LIN {X 0,Y 488.682,Z 691.608,A -85,B 0,C 180,E1 -6498.445,E2 -6498.445} C_VEL
LIN {X 0,Y 488.641,Z 691.61,A -85,B 0,C 180,E1 -6501.074,E2 -6501.074} C_VEL
LIN {X 0,Y 488.644,Z 691.62,A -85,B 0,C 180,E1 -6503.748,E2 -6503.748} C_VEL
LIN {X 0,Y 488.702,Z 691.604,A -85,B 0,C 180,E1 -6506.475,E2 -6506.475} C_VEL
LIN {X 0,Y 488.669,Z 691.61,A -85,B 0,C 180,E1 -6509.274,E2 -6509.274} C_VEL
LIN {X 0,Y 488.646,Z 691.618,A -85,B 0,C 180,E1 -6512.151,E2 -6512.151} C_VEL
LIN {X 0,Y 488.663,Z 691.609,A -85,B 0,C 180,E1 -6515.12,E2 -6515.12} C_VEL
LIN {X 0,Y 488.636,Z 691.613,A -85,B 0,C 180,E1 -6518.204,E2 -6518.204} C_VEL
LIN {X 0,Y 488.696,Z 691.613,A -85,B 0,C 180,E1 -6520.355,E2 -6520.355} C_VEL
LIN {X 0,Y 488.667,Z 691.611,A -85,B 0,C 180,E1 -6523.657,E2 -6523.657} C_VEL
LIN {X 0,Y 488.67,Z 691.617,A -85,B 0,C 180,E1 -6526.355,E2 -6526.355} C_VEL
LIN {X 0,Y 488.691,Z 691.609,A -85,B 0,C 180,E1 -6529.683,E2 -6529.683} C_VEL
LIN {X 0,Y 488.64,Z 691.619,A -85,B 0,C 180,E1 -6532.284,E2 -6532.284} C_VEL
LIN {X 0,Y 488.691,Z 691.608,A -85,B 0,C 180,E1 -6535.058,E2 -6535.058} C_VEL
LIN {X 0,Y 488.671,Z 691.615,A -85,B 0,C 180,E1 -6538.052,E2 -6538.052} C_VEL
LIN {X 0,Y 488.749,Z 691.808,A -85,B 0,C 180,E1 -6540.178,E2 -6540.178} C_VEL
LIN {X 0,Y 492.403,Z 708.291,A -85,B 0,C 180,E1 -6542.534,E2 -6542.534} C_VEL
LIN {X 0,Y 491.834,Z 726.438,A -85,B 0,C 180,E1 -6544.85,E2 -6544.85} C_VEL
LIN {X 0,Y 491.007,Z 751.019,A -85,B 0,C 180,E1 -6547.938,E2 -6547.938} C_VEL
LIN {X 0,Y 490.21,Z 776.598,A -85,B 0,C 180,E1 -6551.125,E2 -6551.125} C_VEL
LIN {X 0,Y 489.614,Z 797.522,A -85,B 0,C 180,E1 -6553.716,E2 -6553.716} C_VEL
LIN {X 0,Y 491.626,Z 815.137,A -85,B 0,C 180,E1 -6554.041,E2 -6554.041} C_VEL
LIN {X 0,Y 491.033,Z 908.334,A -85,B 0,C 180,E1 -6555.422,E2 -6555.422} C_VEL
LIN {X 0,Y 490.681,Z 921.584,A -85,B 0,C 180,E1 -6555.782,E2 -6555.782} C_VEL
LIN {X 0,Y 490.274,Z 934.931,A -85,B 0,C 180,E1 -6556.325,E2 -6556.325} C_VEL
LIN {X 0,Y 489.962,Z 946.2,A -85,B 0,C 180,E1 -6556.95,E2 -6556.95} C_VEL
LIN {X 0,Y 489.582,Z 957.937,A -85,B 0,C 180,E1 -6557.782,E2 -6557.782} C_VEL
LIN {X 0,Y 489.117,Z 968.518,A -85,B 0,C 180,E1 -6558.716,E2 -6558.716} C_VEL
LIN {X 0,Y 488.829,Z 977.207,A -85,B 0,C 180,E1 -6559.653,E2 -6559.653} C_VEL
LIN {X 0,Y 488.559,Z 985.239,A -85,B 0,C 180,E1 -6560.693,E2 -6560.693} C_VEL
LIN {X 0,Y 488.333,Z 993.106,A -85,B 0,C 180,E1 -6561.94,E2 -6561.94} C_VEL
LIN {X 0,Y 488.136,Z 1000.365,A -85,B 0,C 180,E1 -6563.392,E2 -6563.392} C_VEL
LIN {X 0,Y 488.09,Z 1005.213,A -85,B 0,C 180,E1 -6564.636,E2 -6564.636} C_VEL
LIN {X 0,Y 488.029,Z 1008.92,A -85,B 0,C 180,E1 -6565.877,E2 -6565.877} C_VEL
LIN {X 0,Y 488.027,Z 1010.835,A -85,B 0,C 180,E1 -6566.703,E2 -6566.703} C_VEL
LIN {X 0,Y 487.976,Z 1012.263,A -85,B 0,C 180,E1 -6567.529,E2 -6567.529} C_VEL
LIN {X 0,Y 487.951,Z 1013.283,A -85,B 0,C 180,E1 -6568.355,E2 -6568.355} C_VEL
LIN {X 0,Y 487.913,Z 1013.9,A -85,B 0,C 180,E1 -6569.18,E2 -6569.18} C_VEL
LIN {X 0,Y 487.905,Z 1014.118,A -85,B 0,C 180,E1 -6570.005,E2 -6570.005} C_VEL
LIN {X 0,Y 487.913,Z 1013.893,A -85,B 0,C 180,E1 -6570.831,E2 -6570.831} C_VEL
LIN {X 0,Y 487.952,Z 1013.27,A -85,B 0,C 180,E1 -6571.656,E2 -6571.656} C_VEL
LIN {X 0,Y 487.978,Z 1012.245,A -85,B 0,C 180,E1 -6572.482,E2 -6572.482} C_VEL
LIN {X 0,Y 488.03,Z 1010.81,A -85,B 0,C 180,E1 -6573.307,E2 -6573.307} C_VEL
LIN {X 0,Y 488.022,Z 1007.785,A -85,B 0,C 180,E1 -6574.548,E2 -6574.548} C_VEL
LIN {X 0,Y 488.16,Z 1002.71,A -85,B 0,C 180,E1 -6576.045,E2 -6576.045} C_VEL
LIN {X 0,Y 488.241,Z 996.389,A -85,B 0,C 180,E1 -6577.449,E2 -6577.449} C_VEL
LIN {X 0,Y 488.462,Z 989.326,A -85,B 0,C 180,E1 -6578.694,E2 -6578.694} C_VEL
LIN {X 0,Y 488.713,Z 980.494,A -85,B 0,C 180,E1 -6579.942,E2 -6579.942} C_VEL
LIN {X 0,Y 489.054,Z 971.474,A -85,B 0,C 180,E1 -6580.982,E2 -6580.982} C_VEL
LIN {X 0,Y 489.494,Z 960.399,A -85,B 0,C 180,E1 -6582.021,E2 -6582.021} C_VEL
LIN {X 0,Y 489.843,Z 949.728,A -85,B 0,C 180,E1 -6582.821,E2 -6582.821} C_VEL
LIN {X 0,Y 490.162,Z 937.757,A -85,B 0,C 180,E1 -6583.531,E2 -6583.531} C_VEL
LIN {X 0,Y 490.558,Z 924.976,A -85,B 0,C 180,E1 -6584.101,E2 -6584.101} C_VEL
LIN {X 0,Y 490.92,Z 912.426,A -85,B 0,C 180,E1 -6584.487,E2 -6584.487} C_VEL
LIN {X 0,Y 491.114,Z 896.461,A -85,B 0,C 180,E1 -6584.772,E2 -6584.772} C_VEL
LIN {X 0,Y 491.597,Z 814.634,A -85,B 0,C 180,E1 -6585.967,E2 -6585.967} C_VEL
LIN {X 0,Y 489.604,Z 797.347,A -85,B 0,C 180,E1 -6586.302,E2 -6586.302} C_VEL
LIN {X 0,Y 490.277,Z 773.565,A -85,B 0,C 180,E1 -6589.255,E2 -6589.255} C_VEL
LIN {X 0,Y 491.138,Z 747.424,A -85,B 0,C 180,E1 -6592.51,E2 -6592.51} C_VEL
LIN {X 0,Y 491.835,Z 726.347,A -85,B 0,C 180,E1 -6595.162,E2 -6595.162} C_VEL
LIN {X 0,Y 492.39,Z 707.801,A -85,B 0,C 180,E1 -6597.53,E2 -6597.53} C_VEL
LIN {X 0,Y 488.675,Z 691.615,A -85,B 0,C 180,E1 -6599.87,E2 -6599.87} C_VEL
LIN {X 0,Y 488.684,Z 691.608,A -85,B 0,C 180,E1 -6602.152,E2 -6602.152} C_VEL
LIN {X 0,Y 488.637,Z 691.615,A -85,B 0,C 180,E1 -6605.126,E2 -6605.126} C_VEL
LIN {X 0,Y 488.654,Z 691.613,A -85,B 0,C 180,E1 -6608.206,E2 -6608.206} C_VEL
LIN {X 0,Y 488.657,Z 691.617,A -85,B 0,C 180,E1 -6611.425,E2 -6611.425} C_VEL
LIN {X 0,Y 488.711,Z 691.608,A -85,B 0,C 180,E1 -6614.805,E2 -6614.805} C_VEL
LIN {X 0,Y 488.663,Z 691.616,A -85,B 0,C 180,E1 -6617.471,E2 -6617.471} C_VEL
LIN {X 0,Y 488.719,Z 691.607,A -85,B 0,C 180,E1 -6619.675,E2 -6619.675} C_VEL
LIN {X 0,Y 488.673,Z 691.613,A -85,B 0,C 180,E1 -6622.84,E2 -6622.84} C_VEL
LIN {X 0,Y 488.734,Z 691.603,A -85,B 0,C 180,E1 -6625.887,E2 -6625.887} C_VEL
LIN {X 0,Y 488.704,Z 691.608,A -85,B 0,C 180,E1 -6628.821,E2 -6628.821} C_VEL
LIN {X 0,Y 488.712,Z 691.61,A -85,B 0,C 180,E1 -6631.669,E2 -6631.669} C_VEL
LIN {X 0,Y 488.713,Z 691.606,A -85,B 0,C 180,E1 -6634.442,E2 -6634.442} C_VEL
LIN {X 0,Y 488.734,Z 691.609,A -85,B 0,C 180,E1 -6637.154,E2 -6637.154} C_VEL
LIN {X 0,Y 488.737,Z 691.608,A -85,B 0,C 180,E1 -6639.811,E2 -6639.811} C_VEL
LIN {X 0,Y 488.724,Z 691.606,A -85,B 0,C 180,E1 -6642.423,E2 -6642.423} C_VEL
LIN {X 0,Y 488.782,Z 691.601,A -85,B 0,C 180,E1 -6644.316,E2 -6644.316} C_VEL
LIN {X 0,Y 491.379,Z 699.537,A -85,B 0,C 180,E1 -6644.546,E2 -6644.546} C_VEL
LIN {X 0,Y 490.914,Z 771.943,A -85,B 0,C 180,E1 -6645.729,E2 -6645.729} C_VEL
LIN {X 0,Y 490.85,Z 783.407,A -85,B 0,C 180,E1 -6646.044,E2 -6646.044} C_VEL
LIN {X 0,Y 490.738,Z 793.546,A -85,B 0,C 180,E1 -6646.437,E2 -6646.437} C_VEL
LIN {X 0,Y 490.525,Z 803.477,A -85,B 0,C 180,E1 -6646.936,E2 -6646.936} C_VEL
LIN {X 0,Y 490.338,Z 812.486,A -85,B 0,C 180,E1 -6647.5,E2 -6647.5} C_VEL
LIN {X 0,Y 490.066,Z 821.742,A -85,B 0,C 180,E1 -6648.208,E2 -6648.208} C_VEL
LIN {X 0,Y 489.791,Z 830.671,A -85,B 0,C 180,E1 -6649.04,E2 -6649.04} C_VEL
LIN {X 0,Y 489.536,Z 838.156,A -85,B 0,C 180,E1 -6649.871,E2 -6649.871} C_VEL
LIN {X 0,Y 489.241,Z 845.904,A -85,B 0,C 180,E1 -6650.908,E2 -6650.908} C_VEL
LIN {X 0,Y 489.033,Z 852.313,A -85,B 0,C 180,E1 -6651.945,E2 -6651.945} C_VEL
LIN {X 0,Y 488.829,Z 858.14,A -85,B 0,C 180,E1 -6653.095,E2 -6653.095} C_VEL
LIN {X 0,Y 488.697,Z 862.749,A -85,B 0,C 180,E1 -6654.222,E2 -6654.222} C_VEL
LIN {X 0,Y 488.536,Z 865.607,A -85,B 0,C 180,E1 -6655.048,E2 -6655.048} C_VEL
LIN {X 0,Y 488.424,Z 869.61,A -85,B 0,C 180,E1 -6656.7,E2 -6656.7} C_VEL
LIN {X 0,Y 488.434,Z 871.082,A -85,B 0,C 180,E1 -6657.526,E2 -6657.526} C_VEL
LIN {X 0,Y 488.379,Z 872.611,A -85,B 0,C 180,E1 -6659.175,E2 -6659.175} C_VEL
LIN {X 0,Y 488.346,Z 872.803,A -85,B 0,C 180,E1 -6660,E2 -6660} C_VEL
LIN {X 0,Y 488.322,Z 872.573,A -85,B 0,C 180,E1 -6660.825,E2 -6660.825} C_VEL
LIN {X 0,Y 488.287,Z 870.905,A -85,B 0,C 180,E1 -6662.475,E2 -6662.475} C_VEL
LIN {X 0,Y 488.448,Z 867.553,A -85,B 0,C 180,E1 -6664.126,E2 -6664.126} C_VEL
LIN {X 0,Y 488.527,Z 863.892,A -85,B 0,C 180,E1 -6665.366,E2 -6665.366} C_VEL
LIN {X 0,Y 488.748,Z 859.084,A -85,B 0,C 180,E1 -6666.606,E2 -6666.606} C_VEL
LIN {X 0,Y 488.857,Z 854.178,A -85,B 0,C 180,E1 -6667.642,E2 -6667.642} C_VEL
LIN {X 0,Y 489.102,Z 848.229,A -85,B 0,C 180,E1 -6668.678,E2 -6668.678} C_VEL
LIN {X 0,Y 489.325,Z 841.043,A -85,B 0,C 180,E1 -6669.716,E2 -6669.716} C_VEL
LIN {X 0,Y 489.586,Z 832.308,A -85,B 0,C 180,E1 -6670.755,E2 -6670.755} C_VEL
LIN {X 0,Y 489.9,Z 823.903,A -85,B 0,C 180,E1 -6671.586,E2 -6671.586} C_VEL
LIN {X 0,Y 490.138,Z 815.105,A -85,B 0,C 180,E1 -6672.315,E2 -6672.315} C_VEL
LIN {X 0,Y 490.391,Z 805.826,A -85,B 0,C 180,E1 -6672.95,E2 -6672.95} C_VEL
LIN {X 0,Y 490.643,Z 795.612,A -85,B 0,C 180,E1 -6673.513,E2 -6673.513} C_VEL
LIN {X 0,Y 490.802,Z 785.306,A -85,B 0,C 180,E1 -6673.957,E2 -6673.957} C_VEL
LIN {X 0,Y 490.895,Z 774.608,A -85,B 0,C 180,E1 -6674.298,E2 -6674.298} C_VEL
LIN {X 0,Y 491.019,Z 762.121,A -85,B 0,C 180,E1 -6674.559,E2 -6674.559} C_VEL
LIN {X 0,Y 491.415,Z 699.602,A -85,B 0,C 180,E1 -6675.532,E2 -6675.532} C_VEL
LIN {X 0,Y 488.767,Z 691.601,A -85,B 0,C 180,E1 -6675.76,E2 -6675.76} C_VEL
LIN {X 0,Y 488.76,Z 691.604,A -85,B 0,C 180,E1 -6678.442,E2 -6678.442} C_VEL
LIN {X 0,Y 488.72,Z 691.607,A -85,B 0,C 180,E1 -6681.07,E2 -6681.07} C_VEL
LIN {X 0,Y 488.685,Z 691.607,A -85,B 0,C 180,E1 -6683.746,E2 -6683.746} C_VEL
LIN {X 0,Y 488.728,Z 691.609,A -85,B 0,C 180,E1 -6686.925,E2 -6686.925} C_VEL
LIN {X 0,Y 488.737,Z 691.602,A -85,B 0,C 180,E1 -6690.219,E2 -6690.219} C_VEL
LIN {X 0,Y 488.725,Z 691.603,A -85,B 0,C 180,E1 -6693.478,E2 -6693.478} C_VEL
LIN {X 0,Y 488.687,Z 691.608,A -85,B 0,C 180,E1 -6696.351,E2 -6696.351} C_VEL
LIN {X 0,Y 488.708,Z 691.608,A -85,B 0,C 180,E1 -6699.254,E2 -6699.254} C_VEL
LIN {X 0,Y 488.683,Z 691.608,A -85,B 0,C 180,E1 -6702.527,E2 -6702.527} C_VEL
LIN {X 0,Y 488.713,Z 691.609,A -85,B 0,C 180,E1 -6705.195,E2 -6705.195} C_VEL
LIN {X 0,Y 488.677,Z 691.609,A -85,B 0,C 180,E1 -6708.577,E2 -6708.577} C_VEL
LIN {X 0,Y 488.7,Z 691.61,A -85,B 0,C 180,E1 -6710.948,E2 -6710.948} C_VEL
LIN {X 0,Y 488.651,Z 691.611,A -85,B 0,C 180,E1 -6713.447,E2 -6713.447} C_VEL
LIN {X 0,Y 488.007,Z 691.694,A -85,B 0,C 180,E1 -6714.134,E2 -6714.134} C_VEL
LIN {X 0,Y 485.168,Z 692.051,A -85,B 0,C 180,E1 -6715.251,E2 -6715.251} C_VEL
LIN {X 0,Y 482.758,Z 692.346,A -85,B 0,C 180,E1 -6716.152,E2 -6716.152} C_VEL
LIN {X 0,Y 481.726,Z 692.477,A -85,B 0,C 180,E1 -6716.847,E2 -6716.847} C_VEL
LIN {X 0,Y 481.644,Z 692.487,A -85,B 0,C 180,E1 -6717.083,E2 -6717.083} C_VEL
LIN {X 0,Y 481.613,Z 692.487,A -85,B 0,C 180,E1 -6720.25,E2 -6720.25} C_VEL
LIN {X 0,Y 481.642,Z 692.49,A -85,B 0,C 180,E1 -6723.102,E2 -6723.102} C_VEL
LIN {X 0,Y 481.633,Z 692.488,A -85,B 0,C 180,E1 -6725.88,E2 -6725.88} C_VEL
LIN {X 0,Y 481.666,Z 692.488,A -85,B 0,C 180,E1 -6729.04,E2 -6729.04} C_VEL
LIN {X 0,Y 481.665,Z 692.486,A -85,B 0,C 180,E1 -6732.152,E2 -6732.152} C_VEL
LIN {X 0,Y 481.658,Z 692.489,A -85,B 0,C 180,E1 -6733.9,E2 -6733.9} C_VEL
LIN {X 0,Y 485.021,Z 702.116,A -85,B 0,C 180,E1 -6734.18,E2 -6734.18} C_VEL
LIN {X 0,Y 484.543,Z 773.549,A -85,B 0,C 180,E1 -6735.264,E2 -6735.264} C_VEL
LIN {X 0,Y 484.601,Z 786.67,A -85,B 0,C 180,E1 -6735.642,E2 -6735.642} C_VEL
LIN {X 0,Y 484.417,Z 798.704,A -85,B 0,C 180,E1 -6736.146,E2 -6736.146} C_VEL
LIN {X 0,Y 484.157,Z 810.293,A -85,B 0,C 180,E1 -6736.798,E2 -6736.798} C_VEL
LIN {X 0,Y 483.754,Z 821.579,A -85,B 0,C 180,E1 -6737.621,E2 -6737.621} C_VEL
LIN {X 0,Y 483.388,Z 831.928,A -85,B 0,C 180,E1 -6738.57,E2 -6738.57} C_VEL
LIN {X 0,Y 483.057,Z 840.367,A -85,B 0,C 180,E1 -6739.517,E2 -6739.517} C_VEL
LIN {X 0,Y 482.687,Z 848.134,A -85,B 0,C 180,E1 -6740.567,E2 -6740.567} C_VEL
LIN {X 0,Y 482.29,Z 855.831,A -85,B 0,C 180,E1 -6741.848,E2 -6741.848} C_VEL
LIN {X 0,Y 482.153,Z 861.483,A -85,B 0,C 180,E1 -6743.022,E2 -6743.022} C_VEL
LIN {X 0,Y 481.851,Z 867.263,A -85,B 0,C 180,E1 -6744.555,E2 -6744.555} C_VEL
LIN {X 0,Y 481.625,Z 870.803,A -85,B 0,C 180,E1 -6745.811,E2 -6745.811} C_VEL
LIN {X 0,Y 481.532,Z 872.63,A -85,B 0,C 180,E1 -6746.648,E2 -6746.648} C_VEL
LIN {X 0,Y 481.529,Z 874.001,A -85,B 0,C 180,E1 -6747.485,E2 -6747.485} C_VEL
LIN {X 0,Y 481.486,Z 875.581,A -85,B 0,C 180,E1 -6749.158,E2 -6749.158} C_VEL
LIN {X 0,Y 481.469,Z 875.817,A -85,B 0,C 180,E1 -6749.994,E2 -6749.994} C_VEL
LIN {X 0,Y 481.565,Z 875.065,A -85,B 0,C 180,E1 -6751.667,E2 -6751.667} C_VEL
LIN {X 0,Y 481.523,Z 872.825,A -85,B 0,C 180,E1 -6753.341,E2 -6753.341} C_VEL
LIN {X 0,Y 481.685,Z 870.022,A -85,B 0,C 180,E1 -6754.597,E2 -6754.597} C_VEL
LIN {X 0,Y 481.908,Z 866.215,A -85,B 0,C 180,E1 -6755.853,E2 -6755.853} C_VEL
LIN {X 0,Y 482.113,Z 860.745,A -85,B 0,C 180,E1 -6757.242,E2 -6757.242} C_VEL
LIN {X 0,Y 482.412,Z 853.941,A -85,B 0,C 180,E1 -6758.582,E2 -6758.582} C_VEL
LIN {X 0,Y 482.814,Z 845.931,A -85,B 0,C 180,E1 -6759.842,E2 -6759.842} C_VEL
LIN {X 0,Y 483.164,Z 837.724,A -85,B 0,C 180,E1 -6760.894,E2 -6760.894} C_VEL
LIN {X 0,Y 483.542,Z 827.573,A -85,B 0,C 180,E1 -6761.947,E2 -6761.947} C_VEL
LIN {X 0,Y 484.001,Z 817.128,A -85,B 0,C 180,E1 -6762.814,E2 -6762.814} C_VEL
LIN {X 0,Y 484.302,Z 805.369,A -85,B 0,C 180,E1 -6763.592,E2 -6763.592} C_VEL
LIN {X 0,Y 484.494,Z 792.885,A -85,B 0,C 180,E1 -6764.211,E2 -6764.211} C_VEL
LIN {X 0,Y 484.657,Z 779.801,A -85,B 0,C 180,E1 -6764.667,E2 -6764.667} C_VEL
LIN {X 0,Y 484.662,Z 767.477,A -85,B 0,C 180,E1 -6764.935,E2 -6764.935} C_VEL
LIN {X 0,Y 485.002,Z 701.859,A -85,B 0,C 180,E1 -6765.916,E2 -6765.916} C_VEL
LIN {X 0,Y 481.693,Z 692.485,A -85,B 0,C 180,E1 -6766.185,E2 -6766.185} C_VEL
LIN {X 0,Y 481.693,Z 692.488,A -85,B 0,C 180,E1 -6768.715,E2 -6768.715} C_VEL
LIN {X 0,Y 481.626,Z 692.489,A -85,B 0,C 180,E1 -6771.388,E2 -6771.388} C_VEL
LIN {X 0,Y 481.628,Z 692.485,A -85,B 0,C 180,E1 -6774.108,E2 -6774.108} C_VEL
LIN {X 0,Y 481.689,Z 692.485,A -85,B 0,C 180,E1 -6777.125,E2 -6777.125} C_VEL
LIN {X 0,Y 481.649,Z 692.485,A -85,B 0,C 180,E1 -6779.734,E2 -6779.734} C_VEL
LIN {X 0,Y 481.639,Z 692.487,A -85,B 0,C 180,E1 -6782.668,E2 -6782.668} C_VEL
LIN {X 0,Y 481.605,Z 692.494,A -85,B 0,C 180,E1 -6785.703,E2 -6785.703} C_VEL
LIN {X 0,Y 481.673,Z 692.48,A -85,B 0,C 180,E1 -6789.347,E2 -6789.347} C_VEL
LIN {X 0,Y 481.631,Z 692.489,A -85,B 0,C 180,E1 -6792.151,E2 -6792.151} C_VEL
LIN {X 0,Y 481.613,Z 692.482,A -85,B 0,C 180,E1 -6794.451,E2 -6794.451} C_VEL
LIN {X 0,Y 481.639,Z 692.482,A -85,B 0,C 180,E1 -6796.84,E2 -6796.84} C_VEL
LIN {X 0,Y 481.661,Z 692.486,A -85,B 0,C 180,E1 -6800.058,E2 -6800.058} C_VEL
LIN {X 0,Y 481.574,Z 692.495,A -85,B 0,C 180,E1 -6803.37,E2 -6803.37} C_VEL
LIN {X 0,Y 481.649,Z 692.487,A -85,B 0,C 180,E1 -6806.325,E2 -6806.325} C_VEL
LIN {X 0,Y 481.6,Z 692.49,A -85,B 0,C 180,E1 -6809.41,E2 -6809.41} C_VEL
LIN {X 0,Y 481.637,Z 692.49,A -85,B 0,C 180,E1 -6812.164,E2 -6812.164} C_VEL
LIN {X 0,Y 481.653,Z 692.482,A -85,B 0,C 180,E1 -6814.966,E2 -6814.966} C_VEL
LIN {X 0,Y 481.585,Z 692.49,A -85,B 0,C 180,E1 -6817.701,E2 -6817.701} C_VEL
LIN {X 0,Y 481.636,Z 692.493,A -85,B 0,C 180,E1 -6820.39,E2 -6820.39} C_VEL
LIN {X 0,Y 481.621,Z 692.486,A -85,B 0,C 180,E1 -6823.031,E2 -6823.031} C_VEL
LIN {X 0,Y 481.631,Z 692.486,A -85,B 0,C 180,E1 -6825.637,E2 -6825.637} C_VEL
LIN {X 0,Y 481.723,Z 692.477,A -85,B 0,C 180,E1 -6828.214,E2 -6828.214} C_VEL
LIN {X 0,Y 481.695,Z 692.479,A -85,B 0,C 180,E1 -6831.61,E2 -6831.61} C_VEL
LIN {X 0,Y 481.756,Z 692.472,A -85,B 0,C 180,E1 -6834.139,E2 -6834.139} C_VEL
LIN {X 0,Y 481.859,Z 692.46,A -85,B 0,C 180,E1 -6837.492,E2 -6837.492} C_VEL
LIN {X 0,Y 481.859,Z 692.459,A -85,B 0,C 180,E1 -6840,E2 -6840} C_VEL
LIN {X 0,Y 481.859,Z 692.457,A -85,B 0,C 180,E1 -6842.508,E2 -6842.508} C_VEL
LIN {X 0,Y 481.756,Z 692.473,A -85,B 0,C 180,E1 -6845.861,E2 -6845.861} C_VEL
LIN {X 0,Y 481.695,Z 692.476,A -85,B 0,C 180,E1 -6848.389,E2 -6848.389} C_VEL
LIN {X 0,Y 481.722,Z 692.478,A -85,B 0,C 180,E1 -6851.786,E2 -6851.786} C_VEL
LIN {X 0,Y 481.675,Z 692.486,A -85,B 0,C 180,E1 -6855.226,E2 -6855.226} C_VEL
LIN {X 0,Y 481.64,Z 692.485,A -85,B 0,C 180,E1 -6858.725,E2 -6858.725} C_VEL
LIN {X 0,Y 481.583,Z 692.493,A -85,B 0,C 180,E1 -6861.398,E2 -6861.398} C_VEL
LIN {X 0,Y 481.627,Z 692.488,A -85,B 0,C 180,E1 -6864.116,E2 -6864.116} C_VEL
LIN {X 0,Y 481.686,Z 692.478,A -85,B 0,C 180,E1 -6867.145,E2 -6867.145} C_VEL
LIN {X 0,Y 481.626,Z 692.493,A -85,B 0,C 180,E1 -6869.745,E2 -6869.745} C_VEL
LIN {X 0,Y 481.613,Z 692.489,A -85,B 0,C 180,E1 -6872.679,E2 -6872.679} C_VEL
LIN {X 0,Y 481.584,Z 692.495,A -85,B 0,C 180,E1 -6875.714,E2 -6875.714} C_VEL
LIN {X 0,Y 481.673,Z 692.475,A -85,B 0,C 180,E1 -6879.361,E2 -6879.361} C_VEL
LIN {X 0,Y 481.624,Z 692.495,A -85,B 0,C 180,E1 -6882.163,E2 -6882.163} C_VEL
LIN {X 0,Y 481.611,Z 692.495,A -85,B 0,C 180,E1 -6884.463,E2 -6884.463} C_VEL
LIN {X 0,Y 481.643,Z 692.484,A -85,B 0,C 180,E1 -6886.852,E2 -6886.852} C_VEL
LIN {X 0,Y 481.647,Z 692.489,A -85,B 0,C 180,E1 -6890.067,E2 -6890.067} C_VEL
LIN {X 0,Y 481.589,Z 692.493,A -85,B 0,C 180,E1 -6893.26,E2 -6893.26} C_VEL
LIN {X 0,Y 481.675,Z 692.478,A -85,B 0,C 180,E1 -6896.337,E2 -6896.337} C_VEL
LIN {X 0,Y 481.714,Z 692.67,A -85,B 0,C 180,E1 -6899.939,E2 -6899.939} C_VEL
LIN {X 0,Y 485.499,Z 709.671,A -85,B 0,C 180,E1 -6902.413,E2 -6902.413} C_VEL
LIN {X 0,Y 484.924,Z 727.286,A -85,B 0,C 180,E1 -6904.696,E2 -6904.696} C_VEL
LIN {X 0,Y 484.001,Z 753.142,A -85,B 0,C 180,E1 -6907.992,E2 -6907.992} C_VEL
LIN {X 0,Y 483.107,Z 779.604,A -85,B 0,C 180,E1 -6911.342,E2 -6911.342} C_VEL
LIN {X 0,Y 482.611,Z 796.441,A -85,B 0,C 180,E1 -6913.466,E2 -6913.466} C_VEL
LIN {X 0,Y 484.76,Z 816.114,A -85,B 0,C 180,E1 -6913.839,E2 -6913.839} C_VEL
LIN {X 0,Y 484.146,Z 907.318,A -85,B 0,C 180,E1 -6915.21,E2 -6915.21} C_VEL
LIN {X 0,Y 483.776,Z 920.567,A -85,B 0,C 180,E1 -6915.574,E2 -6915.574} C_VEL
LIN {X 0,Y 483.344,Z 933.913,A -85,B 0,C 180,E1 -6916.125,E2 -6916.125} C_VEL
LIN {X 0,Y 482.958,Z 945.493,A -85,B 0,C 180,E1 -6916.778,E2 -6916.778} C_VEL
LIN {X 0,Y 482.547,Z 957.589,A -85,B 0,C 180,E1 -6917.656,E2 -6917.656} C_VEL
LIN {X 0,Y 482.037,Z 968.556,A -85,B 0,C 180,E1 -6918.655,E2 -6918.655} C_VEL
LIN {X 0,Y 481.721,Z 977.898,A -85,B 0,C 180,E1 -6919.711,E2 -6919.711} C_VEL
LIN {X 0,Y 481.42,Z 987.018,A -85,B 0,C 180,E1 -6920.977,E2 -6920.977} C_VEL
LIN {X 0,Y 481.206,Z 994.377,A -85,B 0,C 180,E1 -6922.242,E2 -6922.242} C_VEL
LIN {X 0,Y 481.07,Z 1001.048,A -85,B 0,C 180,E1 -6923.704,E2 -6923.704} C_VEL
LIN {X 0,Y 480.997,Z 1005.548,A -85,B 0,C 180,E1 -6924.976,E2 -6924.976} C_VEL
LIN {X 0,Y 480.974,Z 1007.911,A -85,B 0,C 180,E1 -6925.816,E2 -6925.816} C_VEL
LIN {X 0,Y 480.982,Z 1009.828,A -85,B 0,C 180,E1 -6926.655,E2 -6926.655} C_VEL
LIN {X 0,Y 480.938,Z 1011.258,A -85,B 0,C 180,E1 -6927.493,E2 -6927.493} C_VEL
LIN {X 0,Y 480.916,Z 1012.279,A -85,B 0,C 180,E1 -6928.331,E2 -6928.331} C_VEL
LIN {X 0,Y 480.883,Z 1012.897,A -85,B 0,C 180,E1 -6929.168,E2 -6929.168} C_VEL
LIN {X 0,Y 480.876,Z 1013.115,A -85,B 0,C 180,E1 -6930.006,E2 -6930.006} C_VEL
LIN {X 0,Y 480.883,Z 1012.89,A -85,B 0,C 180,E1 -6930.843,E2 -6930.843} C_VEL
LIN {X 0,Y 480.917,Z 1012.266,A -85,B 0,C 180,E1 -6931.68,E2 -6931.68} C_VEL
LIN {X 0,Y 480.939,Z 1011.24,A -85,B 0,C 180,E1 -6932.518,E2 -6932.518} C_VEL
LIN {X 0,Y 480.985,Z 1009.803,A -85,B 0,C 180,E1 -6933.356,E2 -6933.356} C_VEL
LIN {X 0,Y 480.977,Z 1006.776,A -85,B 0,C 180,E1 -6934.615,E2 -6934.615} C_VEL
LIN {X 0,Y 481.092,Z 1002.699,A -85,B 0,C 180,E1 -6935.874,E2 -6935.874} C_VEL
LIN {X 0,Y 481.158,Z 996.41,A -85,B 0,C 180,E1 -6937.348,E2 -6937.348} C_VEL
LIN {X 0,Y 481.35,Z 989.569,A -85,B 0,C 180,E1 -6938.612,E2 -6938.612} C_VEL
LIN {X 0,Y 481.597,Z 981.098,A -85,B 0,C 180,E1 -6939.878,E2 -6939.878} C_VEL
LIN {X 0,Y 481.943,Z 972.436,A -85,B 0,C 180,E1 -6940.933,E2 -6940.933} C_VEL
LIN {X 0,Y 482.392,Z 961.768,A -85,B 0,C 180,E1 -6941.987,E2 -6941.987} C_VEL
LIN {X 0,Y 482.828,Z 949.931,A -85,B 0,C 180,E1 -6942.926,E2 -6942.926} C_VEL
LIN {X 0,Y 483.19,Z 937.742,A -85,B 0,C 180,E1 -6943.676,E2 -6943.676} C_VEL
LIN {X 0,Y 483.606,Z 925.269,A -85,B 0,C 180,E1 -6944.254,E2 -6944.254} C_VEL
LIN {X 0,Y 483.995,Z 912.471,A -85,B 0,C 180,E1 -6944.672,E2 -6944.672} C_VEL
LIN {X 0,Y 484.203,Z 899.035,A -85,B 0,C 180,E1 -6944.934,E2 -6944.934} C_VEL
LIN {X 0,Y 484.757,Z 815.001,A -85,B 0,C 180,E1 -6946.178,E2 -6946.178} C_VEL
LIN {X 0,Y 482.58,Z 796.32,A -85,B 0,C 180,E1 -6946.546,E2 -6946.546} C_VEL
LIN {X 0,Y 483.285,Z 773.894,A -85,B 0,C 180,E1 -6949.383,E2 -6949.383} C_VEL
LIN {X 0,Y 484.171,Z 748.254,A -85,B 0,C 180,E1 -6952.627,E2 -6952.627} C_VEL
LIN {X 0,Y 484.929,Z 727.191,A -85,B 0,C 180,E1 -6955.316,E2 -6955.316} C_VEL
LIN {X 0,Y 485.52,Z 709.573,A -85,B 0,C 180,E1 -6957.598,E2 -6957.598} C_VEL
LIN {X 0,Y 481.634,Z 692.492,A -85,B 0,C 180,E1 -6960.11,E2 -6960.11} C_VEL
LIN {X 0,Y 481.626,Z 692.487,A -85,B 0,C 180,E1 -6962.682,E2 -6962.682} C_VEL
LIN {X 0,Y 481.58,Z 692.489,A -85,B 0,C 180,E1 -6965.718,E2 -6965.718} C_VEL
LIN {X 0,Y 481.629,Z 692.492,A -85,B 0,C 180,E1 -6968.867,E2 -6968.867} C_VEL
LIN {X 0,Y 481.624,Z 692.488,A -85,B 0,C 180,E1 -6971.909,E2 -6971.909} C_VEL
LIN {X 0,Y 481.647,Z 692.485,A -85,B 0,C 180,E1 -6974.463,E2 -6974.463} C_VEL
LIN {X 0,Y 481.627,Z 692.49,A -85,B 0,C 180,E1 -6976.858,E2 -6976.858} C_VEL
LIN {X 0,Y 481.671,Z 692.482,A -85,B 0,C 180,E1 -6980.059,E2 -6980.059} C_VEL
LIN {X 0,Y 481.631,Z 692.494,A -85,B 0,C 180,E1 -6983.38,E2 -6983.38} C_VEL
LIN {X 0,Y 481.686,Z 692.48,A -85,B 0,C 180,E1 -6986.328,E2 -6986.328} C_VEL
LIN {X 0,Y 481.662,Z 692.489,A -85,B 0,C 180,E1 -6989.419,E2 -6989.419} C_VEL
LIN {X 0,Y 481.67,Z 692.484,A -85,B 0,C 180,E1 -6992.166,E2 -6992.166} C_VEL
LIN {X 0,Y 481.691,Z 692.484,A -85,B 0,C 180,E1 -6994.968,E2 -6994.968} C_VEL
LIN {X 0,Y 481.661,Z 692.489,A -85,B 0,C 180,E1 -6997.705,E2 -6997.705} C_VEL
LIN {X 0,Y 481.717,Z 692.479,A -85,B 0,C 180,E1 -7000.393,E2 -7000.393} C_VEL
LIN {X 0,Y 481.688,Z 692.486,A -85,B 0,C 180,E1 -7003.034,E2 -7003.034} C_VEL
LIN {X 0,Y 481.727,Z 692.481,A -85,B 0,C 180,E1 -7004.067,E2 -7004.067} C_VEL
LIN {X 0,Y 484.579,Z 700.942,A -85,B 0,C 180,E1 -7004.328,E2 -7004.328} C_VEL
LIN {X 0,Y 484.029,Z 773.443,A -85,B 0,C 180,E1 -7005.549,E2 -7005.549} C_VEL
LIN {X 0,Y 483.946,Z 784.76,A -85,B 0,C 180,E1 -7005.868,E2 -7005.868} C_VEL
LIN {X 0,Y 483.884,Z 795.369,A -85,B 0,C 180,E1 -7006.295,E2 -7006.295} C_VEL
LIN {X 0,Y 483.63,Z 805.455,A -85,B 0,C 180,E1 -7006.819,E2 -7006.819} C_VEL
LIN {X 0,Y 483.414,Z 814.468,A -85,B 0,C 180,E1 -7007.404,E2 -7007.404} C_VEL
LIN {X 0,Y 483.126,Z 823.784,A -85,B 0,C 180,E1 -7008.143,E2 -7008.143} C_VEL
LIN {X 0,Y 482.885,Z 831.592,A -85,B 0,C 180,E1 -7008.881,E2 -7008.881} C_VEL
LIN {X 0,Y 482.615,Z 839.118,A -85,B 0,C 180,E1 -7009.724,E2 -7009.724} C_VEL
LIN {X 0,Y 482.302,Z 846.898,A -85,B 0,C 180,E1 -7010.776,E2 -7010.776} C_VEL
LIN {X 0,Y 482.078,Z 853.333,A -85,B 0,C 180,E1 -7011.828,E2 -7011.828} C_VEL
LIN {X 0,Y 481.877,Z 859.169,A -85,B 0,C 180,E1 -7012.993,E2 -7012.993} C_VEL
LIN {X 0,Y 481.731,Z 863.8,A -85,B 0,C 180,E1 -7014.139,E2 -7014.139} C_VEL
LIN {X 0,Y 481.542,Z 866.665,A -85,B 0,C 180,E1 -7014.976,E2 -7014.976} C_VEL
LIN {X 0,Y 481.416,Z 870.674,A -85,B 0,C 180,E1 -7016.652,E2 -7016.652} C_VEL
LIN {X 0,Y 481.427,Z 872.141,A -85,B 0,C 180,E1 -7017.49,E2 -7017.49} C_VEL
LIN {X 0,Y 481.372,Z 873.659,A -85,B 0,C 180,E1 -7019.163,E2 -7019.163} C_VEL
LIN {X 0,Y 481.339,Z 873.839,A -85,B 0,C 180,E1 -7020,E2 -7020} C_VEL
LIN {X 0,Y 481.32,Z 873.595,A -85,B 0,C 180,E1 -7020.837,E2 -7020.837} C_VEL
LIN {X 0,Y 481.265,Z 871.904,A -85,B 0,C 180,E1 -7022.511,E2 -7022.511} C_VEL
LIN {X 0,Y 481.432,Z 868.506,A -85,B 0,C 180,E1 -7024.186,E2 -7024.186} C_VEL
LIN {X 0,Y 481.528,Z 864.809,A -85,B 0,C 180,E1 -7025.444,E2 -7025.444} C_VEL
LIN {X 0,Y 481.765,Z 859.966,A -85,B 0,C 180,E1 -7026.702,E2 -7026.702} C_VEL
LIN {X 0,Y 481.891,Z 855.009,A -85,B 0,C 180,E1 -7027.753,E2 -7027.753} C_VEL
LIN {X 0,Y 482.125,Z 849.013,A -85,B 0,C 180,E1 -7028.804,E2 -7028.804} C_VEL
LIN {X 0,Y 482.385,Z 841.769,A -85,B 0,C 180,E1 -7029.857,E2 -7029.857} C_VEL
LIN {X 0,Y 482.607,Z 834.946,A -85,B 0,C 180,E1 -7030.7,E2 -7030.7} C_VEL
LIN {X 0,Y 482.934,Z 825.668,A -85,B 0,C 180,E1 -7031.649,E2 -7031.649} C_VEL
LIN {X 0,Y 483.209,Z 817.022,A -85,B 0,C 180,E1 -7032.388,E2 -7032.388} C_VEL
LIN {X 0,Y 483.467,Z 806.876,A -85,B 0,C 180,E1 -7033.098,E2 -7033.098} C_VEL
LIN {X 0,Y 483.718,Z 796.935,A -85,B 0,C 180,E1 -7033.656,E2 -7033.656} C_VEL
LIN {X 0,Y 483.909,Z 786.02,A -85,B 0,C 180,E1 -7034.133,E2 -7034.133} C_VEL
LIN {X 0,Y 484.012,Z 775.252,A -85,B 0,C 180,E1 -7034.479,E2 -7034.479} C_VEL
LIN {X 0,Y 484.133,Z 762.67,A -85,B 0,C 180,E1 -7034.744,E2 -7034.744} C_VEL
LIN {X 0,Y 484.557,Z 701.038,A -85,B 0,C 180,E1 -7035.725,E2 -7035.725} C_VEL
LIN {X 0,Y 481.716,Z 692.48,A -85,B 0,C 180,E1 -7035.979,E2 -7035.979} C_VEL
LIN {X 0,Y 481.721,Z 692.483,A -85,B 0,C 180,E1 -7038.721,E2 -7038.721} C_VEL
LIN {X 0,Y 481.658,Z 692.484,A -85,B 0,C 180,E1 -7041.394,E2 -7041.394} C_VEL
LIN {X 0,Y 481.665,Z 692.483,A -85,B 0,C 180,E1 -7044.114,E2 -7044.114} C_VEL
LIN {X 0,Y 481.7,Z 692.481,A -85,B 0,C 180,E1 -7047.124,E2 -7047.124} C_VEL
LIN {X 0,Y 481.687,Z 692.479,A -85,B 0,C 180,E1 -7049.741,E2 -7049.741} C_VEL
LIN {X 0,Y 481.667,Z 692.487,A -85,B 0,C 180,E1 -7052.675,E2 -7052.675} C_VEL
LIN {X 0,Y 481.645,Z 692.484,A -85,B 0,C 180,E1 -7055.709,E2 -7055.709} C_VEL
LIN {X 0,Y 481.681,Z 692.487,A -85,B 0,C 180,E1 -7058.858,E2 -7058.858} C_VEL
LIN {X 0,Y 481.641,Z 692.483,A -85,B 0,C 180,E1 -7062.162,E2 -7062.162} C_VEL
LIN {X 0,Y 481.67,Z 692.48,A -85,B 0,C 180,E1 -7064.457,E2 -7064.457} C_VEL
LIN {X 0,Y 481.63,Z 692.485,A -85,B 0,C 180,E1 -7067.834,E2 -7067.834} C_VEL
LIN {X 0,Y 481.661,Z 692.483,A -85,B 0,C 180,E1 -7070.654,E2 -7070.654} C_VEL
LIN {X 0,Y 481.617,Z 692.49,A -85,B 0,C 180,E1 -7073.442,E2 -7073.442} C_VEL
LIN {X 0,Y 481.687,Z 692.477,A -85,B 0,C 180,E1 -7076.324,E2 -7076.324} C_VEL
LIN {X 0,Y 481.644,Z 692.487,A -85,B 0,C 180,E1 -7077.083,E2 -7077.083} C_VEL
LIN {X 0,Y 480.979,Z 692.574,A -85,B 0,C 180,E1 -7077.781,E2 -7077.781} C_VEL
LIN {X 0,Y 478.111,Z 692.928,A -85,B 0,C 180,E1 -7078.914,E2 -7078.914} C_VEL
LIN {X 0,Y 475.69,Z 693.226,A -85,B 0,C 180,E1 -7079.827,E2 -7079.827} C_VEL
LIN {X 0,Y 474.662,Z 693.354,A -85,B 0,C 180,E1 -7080.533,E2 -7080.533} C_VEL
LIN {X 0,Y 474.584,Z 693.365,A -85,B 0,C 180,E1 -7080.772,E2 -7080.772} C_VEL
LIN {X 0,Y 474.569,Z 693.37,A -85,B 0,C 180,E1 -7083.619,E2 -7083.619} C_VEL
LIN {X 0,Y 474.611,Z 693.363,A -85,B 0,C 180,E1 -7086.649,E2 -7086.649} C_VEL
LIN {X 0,Y 474.629,Z 693.366,A -85,B 0,C 180,E1 -7089.179,E2 -7089.179} C_VEL
LIN {X 0,Y 474.626,Z 693.364,A -85,B 0,C 180,E1 -7091.879,E2 -7091.879} C_VEL
LIN {X 0,Y 474.615,Z 693.368,A -85,B 0,C 180,E1 -7093.655,E2 -7093.655} C_VEL
LIN {X 0,Y 478.274,Z 704.058,A -85,B 0,C 180,E1 -7093.965,E2 -7093.965} C_VEL
LIN {X 0,Y 477.746,Z 774.571,A -85,B 0,C 180,E1 -7095.05,E2 -7095.05} C_VEL
LIN {X 0,Y 477.794,Z 787.686,A -85,B 0,C 180,E1 -7095.433,E2 -7095.433} C_VEL
LIN {X 0,Y 477.595,Z 799.716,A -85,B 0,C 180,E1 -7095.944,E2 -7095.944} C_VEL
LIN {X 0,Y 477.318,Z 811.297,A -85,B 0,C 180,E1 -7096.605,E2 -7096.605} C_VEL
LIN {X 0,Y 476.893,Z 822.587,A -85,B 0,C 180,E1 -7097.44,E2 -7097.44} C_VEL
LIN {X 0,Y 476.503,Z 832.935,A -85,B 0,C 180,E1 -7098.402,E2 -7098.402} C_VEL
LIN {X 0,Y 476.152,Z 841.373,A -85,B 0,C 180,E1 -7099.363,E2 -7099.363} C_VEL
LIN {X 0,Y 475.759,Z 849.139,A -85,B 0,C 180,E1 -7100.429,E2 -7100.429} C_VEL
LIN {X 0,Y 475.335,Z 856.836,A -85,B 0,C 180,E1 -7101.728,E2 -7101.728} C_VEL
LIN {X 0,Y 475.18,Z 862.486,A -85,B 0,C 180,E1 -7102.919,E2 -7102.919} C_VEL
LIN {X 0,Y 474.865,Z 868.266,A -85,B 0,C 180,E1 -7104.474,E2 -7104.474} C_VEL
LIN {X 0,Y 474.616,Z 871.807,A -85,B 0,C 180,E1 -7105.749,E2 -7105.749} C_VEL
LIN {X 0,Y 474.515,Z 873.633,A -85,B 0,C 180,E1 -7106.598,E2 -7106.598} C_VEL
LIN {X 0,Y 474.514,Z 875.003,A -85,B 0,C 180,E1 -7107.448,E2 -7107.448} C_VEL
LIN {X 0,Y 474.467,Z 876.583,A -85,B 0,C 180,E1 -7109.146,E2 -7109.146} C_VEL
LIN {X 0,Y 474.449,Z 876.818,A -85,B 0,C 180,E1 -7109.994,E2 -7109.994} C_VEL
LIN {X 0,Y 474.551,Z 876.065,A -85,B 0,C 180,E1 -7111.692,E2 -7111.692} C_VEL
LIN {X 0,Y 474.506,Z 873.827,A -85,B 0,C 180,E1 -7113.391,E2 -7113.391} C_VEL
LIN {X 0,Y 474.679,Z 871.023,A -85,B 0,C 180,E1 -7114.665,E2 -7114.665} C_VEL
LIN {X 0,Y 474.925,Z 867.216,A -85,B 0,C 180,E1 -7115.94,E2 -7115.94} C_VEL
LIN {X 0,Y 475.142,Z 861.744,A -85,B 0,C 180,E1 -7117.349,E2 -7117.349} C_VEL
LIN {X 0,Y 475.466,Z 854.941,A -85,B 0,C 180,E1 -7118.708,E2 -7118.708} C_VEL
LIN {X 0,Y 475.894,Z 846.93,A -85,B 0,C 180,E1 -7119.986,E2 -7119.986} C_VEL
LIN {X 0,Y 476.291,Z 838.719,A -85,B 0,C 180,E1 -7121.053,E2 -7121.053} C_VEL
LIN {X 0,Y 476.669,Z 828.571,A -85,B 0,C 180,E1 -7122.122,E2 -7122.122} C_VEL
LIN {X 0,Y 477.15,Z 818.124,A -85,B 0,C 180,E1 -7123.002,E2 -7123.002} C_VEL
LIN {X 0,Y 477.473,Z 806.364,A -85,B 0,C 180,E1 -7123.791,E2 -7123.791} C_VEL
LIN {X 0,Y 477.675,Z 793.879,A -85,B 0,C 180,E1 -7124.418,E2 -7124.418} C_VEL
LIN {X 0,Y 477.844,Z 780.791,A -85,B 0,C 180,E1 -7124.881,E2 -7124.881} C_VEL
LIN {X 0,Y 477.841,Z 768.456,A -85,B 0,C 180,E1 -7125.154,E2 -7125.154} C_VEL
LIN {X 0,Y 478.238,Z 703.504,A -85,B 0,C 180,E1 -7126.137,E2 -7126.137} C_VEL
LIN {X 0,Y 474.629,Z 693.368,A -85,B 0,C 180,E1 -7126.433,E2 -7126.433} C_VEL
LIN {X 0,Y 474.647,Z 693.366,A -85,B 0,C 180,E1 -7129.004,E2 -7129.004} C_VEL
LIN {X 0,Y 474.569,Z 693.366,A -85,B 0,C 180,E1 -7131.722,E2 -7131.722} C_VEL
LIN {X 0,Y 474.606,Z 693.362,A -85,B 0,C 180,E1 -7134.488,E2 -7134.488} C_VEL
LIN {X 0,Y 474.647,Z 693.36,A -85,B 0,C 180,E1 -7137.326,E2 -7137.326} C_VEL
LIN {X 0,Y 474.575,Z 693.364,A -85,B 0,C 180,E1 -7140.223,E2 -7140.223} C_VEL
LIN {X 0,Y 474.61,Z 693.368,A -85,B 0,C 180,E1 -7143.213,E2 -7143.213} C_VEL
LIN {X 0,Y 474.554,Z 693.368,A -85,B 0,C 180,E1 -7146.317,E2 -7146.317} C_VEL
LIN {X 0,Y 474.61,Z 693.366,A -85,B 0,C 180,E1 -7149.644,E2 -7149.644} C_VEL
LIN {X 0,Y 474.607,Z 693.363,A -85,B 0,C 180,E1 -7152.924,E2 -7152.924} C_VEL
LIN {X 0,Y 474.569,Z 693.366,A -85,B 0,C 180,E1 -7155.89,E2 -7155.89} C_VEL
LIN {X 0,Y 474.595,Z 693.364,A -85,B 0,C 180,E1 -7159.032,E2 -7159.032} C_VEL
LIN {X 0,Y 474.566,Z 693.37,A -85,B 0,C 180,E1 -7161.697,E2 -7161.697} C_VEL
LIN {X 0,Y 474.571,Z 693.365,A -85,B 0,C 180,E1 -7164.721,E2 -7164.721} C_VEL
LIN {X 0,Y 474.578,Z 693.368,A -85,B 0,C 180,E1 -7167.783,E2 -7167.783} C_VEL
LIN {X 0,Y 474.567,Z 693.362,A -85,B 0,C 180,E1 -7170.878,E2 -7170.878} C_VEL
LIN {X 0,Y 474.6,Z 693.363,A -85,B 0,C 180,E1 -7173.625,E2 -7173.625} C_VEL
LIN {X 0,Y 474.567,Z 693.367,A -85,B 0,C 180,E1 -7176.637,E2 -7176.637} C_VEL
LIN {X 0,Y 474.585,Z 693.368,A -85,B 0,C 180,E1 -7180.086,E2 -7180.086} C_VEL
LIN {X 0,Y 474.58,Z 693.366,A -85,B 0,C 180,E1 -7182.772,E2 -7182.772} C_VEL
LIN {X 0,Y 474.587,Z 693.364,A -85,B 0,C 180,E1 -7185.419,E2 -7185.419} C_VEL
LIN {X 0,Y 474.665,Z 693.354,A -85,B 0,C 180,E1 -7188.036,E2 -7188.036} C_VEL
LIN {X 0,Y 474.66,Z 693.356,A -85,B 0,C 180,E1 -7191.485,E2 -7191.485} C_VEL
LIN {X 0,Y 474.716,Z 693.349,A -85,B 0,C 180,E1 -7194.052,E2 -7194.052} C_VEL
LIN {X 0,Y 474.826,Z 693.336,A -85,B 0,C 180,E1 -7197.455,E2 -7197.455} C_VEL
LIN {X 0,Y 474.831,Z 693.335,A -85,B 0,C 180,E1 -7200,E2 -7200} C_VEL
LIN {X 0,Y 474.826,Z 693.333,A -85,B 0,C 180,E1 -7202.545,E2 -7202.545} C_VEL
LIN {X 0,Y 474.716,Z 693.35,A -85,B 0,C 180,E1 -7205.948,E2 -7205.948} C_VEL
LIN {X 0,Y 474.66,Z 693.353,A -85,B 0,C 180,E1 -7208.515,E2 -7208.515} C_VEL
LIN {X 0,Y 474.665,Z 693.356,A -85,B 0,C 180,E1 -7211.963,E2 -7211.963} C_VEL
LIN {X 0,Y 474.63,Z 693.362,A -85,B 0,C 180,E1 -7215.78,E2 -7215.78} C_VEL
LIN {X 0,Y 474.593,Z 693.365,A -85,B 0,C 180,E1 -7219.013,E2 -7219.013} C_VEL
LIN {X 0,Y 474.527,Z 693.375,A -85,B 0,C 180,E1 -7221.732,E2 -7221.732} C_VEL
LIN {X 0,Y 474.607,Z 693.36,A -85,B 0,C 180,E1 -7224.496,E2 -7224.496} C_VEL
LIN {X 0,Y 474.633,Z 693.358,A -85,B 0,C 180,E1 -7227.343,E2 -7227.343} C_VEL
LIN {X 0,Y 474.55,Z 693.366,A -85,B 0,C 180,E1 -7230.817,E2 -7230.817} C_VEL
LIN {X 0,Y 474.578,Z 693.37,A -85,B 0,C 180,E1 -7233.989,E2 -7233.989} C_VEL
LIN {X 0,Y 474.519,Z 693.371,A -85,B 0,C 180,E1 -7236.905,E2 -7236.905} C_VEL
LIN {X 0,Y 474.616,Z 693.355,A -85,B 0,C 180,E1 -7239.659,E2 -7239.659} C_VEL
LIN {X 0,Y 474.602,Z 693.363,A -85,B 0,C 180,E1 -7242.936,E2 -7242.936} C_VEL
LIN {X 0,Y 474.571,Z 693.369,A -85,B 0,C 180,E1 -7245.902,E2 -7245.902} C_VEL
LIN {X 0,Y 474.604,Z 693.365,A -85,B 0,C 180,E1 -7249.044,E2 -7249.044} C_VEL
LIN {X 0,Y 474.576,Z 693.366,A -85,B 0,C 180,E1 -7251.71,E2 -7251.71} C_VEL
LIN {X 0,Y 474.592,Z 693.369,A -85,B 0,C 180,E1 -7254.733,E2 -7254.733} C_VEL
LIN {X 0,Y 474.603,Z 693.367,A -85,B 0,C 180,E1 -7257.794,E2 -7257.794} C_VEL
LIN {X 0,Y 474.633,Z 693.483,A -85,B 0,C 180,E1 -7259.684,E2 -7259.684} C_VEL
LIN {X 0,Y 478.525,Z 710.522,A -85,B 0,C 180,E1 -7262.214,E2 -7262.214} C_VEL
LIN {X 0,Y 478.365,Z 720.389,A -85,B 0,C 180,E1 -7263.527,E2 -7263.527} C_VEL
LIN {X 0,Y 477.215,Z 749.179,A -85,B 0,C 180,E1 -7267.265,E2 -7267.265} C_VEL
LIN {X 0,Y 476.226,Z 775.842,A -85,B 0,C 180,E1 -7270.694,E2 -7270.694} C_VEL
LIN {X 0,Y 475.613,Z 795.82,A -85,B 0,C 180,E1 -7273.229,E2 -7273.229} C_VEL
LIN {X 0,Y 477.913,Z 817.076,A -85,B 0,C 180,E1 -7273.631,E2 -7273.631} C_VEL
LIN {X 0,Y 477.256,Z 906.301,A -85,B 0,C 180,E1 -7274.991,E2 -7274.991} C_VEL
LIN {X 0,Y 476.886,Z 919.551,A -85,B 0,C 180,E1 -7275.361,E2 -7275.361} C_VEL
LIN {X 0,Y 476.435,Z 932.897,A -85,B 0,C 180,E1 -7275.92,E2 -7275.92} C_VEL
LIN {X 0,Y 476.002,Z 944.15,A -85,B 0,C 180,E1 -7276.56,E2 -7276.56} C_VEL
LIN {X 0,Y 475.533,Z 955.91,A -85,B 0,C 180,E1 -7277.418,E2 -7277.418} C_VEL
LIN {X 0,Y 475.082,Z 966.475,A -85,B 0,C 180,E1 -7278.378,E2 -7278.378} C_VEL
LIN {X 0,Y 474.754,Z 975.165,A -85,B 0,C 180,E1 -7279.343,E2 -7279.343} C_VEL
LIN {X 0,Y 474.465,Z 983.2,A -85,B 0,C 180,E1 -7280.414,E2 -7280.414} C_VEL
LIN {X 0,Y 474.19,Z 991.067,A -85,B 0,C 180,E1 -7281.698,E2 -7281.698} C_VEL
LIN {X 0,Y 474.058,Z 996.469,A -85,B 0,C 180,E1 -7282.767,E2 -7282.767} C_VEL
LIN {X 0,Y 474.024,Z 1001.723,A -85,B 0,C 180,E1 -7284.049,E2 -7284.049} C_VEL
LIN {X 0,Y 473.93,Z 1005.799,A -85,B 0,C 180,E1 -7285.328,E2 -7285.328} C_VEL
LIN {X 0,Y 473.938,Z 1008.821,A -85,B 0,C 180,E1 -7286.605,E2 -7286.605} C_VEL
LIN {X 0,Y 473.898,Z 1010.253,A -85,B 0,C 180,E1 -7287.456,E2 -7287.456} C_VEL
LIN {X 0,Y 473.881,Z 1011.274,A -85,B 0,C 180,E1 -7288.306,E2 -7288.306} C_VEL
LIN {X 0,Y 473.853,Z 1011.894,A -85,B 0,C 180,E1 -7289.156,E2 -7289.156} C_VEL
LIN {X 0,Y 473.848,Z 1012.113,A -85,B 0,C 180,E1 -7290.006,E2 -7290.006} C_VEL
LIN {X 0,Y 473.853,Z 1011.887,A -85,B 0,C 180,E1 -7290.855,E2 -7290.855} C_VEL
LIN {X 0,Y 473.882,Z 1011.262,A -85,B 0,C 180,E1 -7291.705,E2 -7291.705} C_VEL
LIN {X 0,Y 473.9,Z 1010.235,A -85,B 0,C 180,E1 -7292.555,E2 -7292.555} C_VEL
LIN {X 0,Y 473.941,Z 1008.796,A -85,B 0,C 180,E1 -7293.406,E2 -7293.406} C_VEL
LIN {X 0,Y 473.934,Z 1005.769,A -85,B 0,C 180,E1 -7294.684,E2 -7294.684} C_VEL
LIN {X 0,Y 474.033,Z 1001.687,A -85,B 0,C 180,E1 -7295.962,E2 -7295.962} C_VEL
LIN {X 0,Y 474.104,Z 995.395,A -85,B 0,C 180,E1 -7297.458,E2 -7297.458} C_VEL
LIN {X 0,Y 474.3,Z 988.552,A -85,B 0,C 180,E1 -7298.741,E2 -7298.741} C_VEL
LIN {X 0,Y 474.541,Z 980.076,A -85,B 0,C 180,E1 -7300.027,E2 -7300.027} C_VEL
LIN {X 0,Y 474.923,Z 971.416,A -85,B 0,C 180,E1 -7301.096,E2 -7301.096} C_VEL
LIN {X 0,Y 475.39,Z 961.005,A -85,B 0,C 180,E1 -7302.143,E2 -7302.143} C_VEL
LIN {X 0,Y 475.801,Z 950.207,A -85,B 0,C 180,E1 -7303.023,E2 -7303.023} C_VEL
LIN {X 0,Y 476.162,Z 938.677,A -85,B 0,C 180,E1 -7303.773,E2 -7303.773} C_VEL
LIN {X 0,Y 476.632,Z 926.875,A -85,B 0,C 180,E1 -7304.358,E2 -7304.358} C_VEL
LIN {X 0,Y 477.07,Z 914.226,A -85,B 0,C 180,E1 -7304.808,E2 -7304.808} C_VEL
LIN {X 0,Y 477.315,Z 901.379,A -85,B 0,C 180,E1 -7305.1,E2 -7305.1} C_VEL
LIN {X 0,Y 477.881,Z 815.191,A -85,B 0,C 180,E1 -7306.399,E2 -7306.399} C_VEL
LIN {X 0,Y 475.583,Z 795.462,A -85,B 0,C 180,E1 -7306.781,E2 -7306.781} C_VEL
LIN {X 0,Y 476.357,Z 771.678,A -85,B 0,C 180,E1 -7309.841,E2 -7309.841} C_VEL
LIN {X 0,Y 477.218,Z 749.073,A -85,B 0,C 180,E1 -7312.747,E2 -7312.747} C_VEL
LIN {X 0,Y 478.054,Z 726.269,A -85,B 0,C 180,E1 -7315.706,E2 -7315.706} C_VEL
LIN {X 0,Y 478.589,Z 710.923,A -85,B 0,C 180,E1 -7317.728,E2 -7317.728} C_VEL
LIN {X 0,Y 474.591,Z 693.37,A -85,B 0,C 180,E1 -7320.354,E2 -7320.354} C_VEL
LIN {X 0,Y 474.58,Z 693.369,A -85,B 0,C 180,E1 -7323.229,E2 -7323.229} C_VEL
LIN {X 0,Y 474.555,Z 693.364,A -85,B 0,C 180,E1 -7326.331,E2 -7326.331} C_VEL
LIN {X 0,Y 474.611,Z 693.365,A -85,B 0,C 180,E1 -7329.553,E2 -7329.553} C_VEL
LIN {X 0,Y 474.58,Z 693.369,A -85,B 0,C 180,E1 -7332.942,E2 -7332.942} C_VEL
LIN {X 0,Y 474.595,Z 693.364,A -85,B 0,C 180,E1 -7335.893,E2 -7335.893} C_VEL
LIN {X 0,Y 474.614,Z 693.365,A -85,B 0,C 180,E1 -7339.047,E2 -7339.047} C_VEL
LIN {X 0,Y 474.607,Z 693.365,A -85,B 0,C 180,E1 -7341.709,E2 -7341.709} C_VEL
LIN {X 0,Y 474.631,Z 693.361,A -85,B 0,C 180,E1 -7344.726,E2 -7344.726} C_VEL
LIN {X 0,Y 474.649,Z 693.359,A -85,B 0,C 180,E1 -7347.789,E2 -7347.789} C_VEL
LIN {X 0,Y 474.616,Z 693.365,A -85,B 0,C 180,E1 -7350.891,E2 -7350.891} C_VEL
LIN {X 0,Y 474.617,Z 693.367,A -85,B 0,C 180,E1 -7353.626,E2 -7353.626} C_VEL
LIN {X 0,Y 474.649,Z 693.359,A -85,B 0,C 180,E1 -7356.643,E2 -7356.643} C_VEL
LIN {X 0,Y 474.667,Z 693.359,A -85,B 0,C 180,E1 -7360.09,E2 -7360.09} C_VEL
LIN {X 0,Y 474.649,Z 693.361,A -85,B 0,C 180,E1 -7362.774,E2 -7362.774} C_VEL
LIN {X 0,Y 474.682,Z 693.359,A -85,B 0,C 180,E1 -7363.815,E2 -7363.815} C_VEL
LIN {X 0,Y 477.806,Z 702.397,A -85,B 0,C 180,E1 -7364.105,E2 -7364.105} C_VEL
LIN {X 0,Y 477.183,Z 774.056,A -85,B 0,C 180,E1 -7365.337,E2 -7365.337} C_VEL
LIN {X 0,Y 477.124,Z 785.536,A -85,B 0,C 180,E1 -7365.662,E2 -7365.662} C_VEL
LIN {X 0,Y 477.036,Z 796.243,A -85,B 0,C 180,E1 -7366.094,E2 -7366.094} C_VEL
LIN {X 0,Y 476.778,Z 806.503,A -85,B 0,C 180,E1 -7366.633,E2 -7366.633} C_VEL
LIN {X 0,Y 476.554,Z 815.455,A -85,B 0,C 180,E1 -7367.22,E2 -7367.22} C_VEL
LIN {X 0,Y 476.245,Z 824.804,A -85,B 0,C 180,E1 -7367.969,E2 -7367.969} C_VEL
LIN {X 0,Y 475.995,Z 832.618,A -85,B 0,C 180,E1 -7368.718,E2 -7368.718} C_VEL
LIN {X 0,Y 475.716,Z 840.148,A -85,B 0,C 180,E1 -7369.573,E2 -7369.573} C_VEL
LIN {X 0,Y 475.393,Z 847.927,A -85,B 0,C 180,E1 -7370.641,E2 -7370.641} C_VEL
LIN {X 0,Y 475.154,Z 854.363,A -85,B 0,C 180,E1 -7371.708,E2 -7371.708} C_VEL
LIN {X 0,Y 474.923,Z 860.122,A -85,B 0,C 180,E1 -7372.87,E2 -7372.87} C_VEL
LIN {X 0,Y 474.762,Z 864.851,A -85,B 0,C 180,E1 -7374.052,E2 -7374.052} C_VEL
LIN {X 0,Y 474.548,Z 867.723,A -85,B 0,C 180,E1 -7374.902,E2 -7374.902} C_VEL
LIN {X 0,Y 474.409,Z 871.737,A -85,B 0,C 180,E1 -7376.603,E2 -7376.603} C_VEL
LIN {X 0,Y 474.42,Z 873.201,A -85,B 0,C 180,E1 -7377.453,E2 -7377.453} C_VEL
LIN {X 0,Y 474.363,Z 874.706,A -85,B 0,C 180,E1 -7379.151,E2 -7379.151} C_VEL
LIN {X 0,Y 474.33,Z 874.877,A -85,B 0,C 180,E1 -7380,E2 -7380} C_VEL
LIN {X 0,Y 474.316,Z 874.619,A -85,B 0,C 180,E1 -7380.849,E2 -7380.849} C_VEL
LIN {X 0,Y 474.243,Z 872.902,A -85,B 0,C 180,E1 -7382.548,E2 -7382.548} C_VEL
LIN {X 0,Y 474.416,Z 869.461,A -85,B 0,C 180,E1 -7384.248,E2 -7384.248} C_VEL
LIN {X 0,Y 474.529,Z 865.726,A -85,B 0,C 180,E1 -7385.524,E2 -7385.524} C_VEL
LIN {X 0,Y 474.784,Z 860.84,A -85,B 0,C 180,E1 -7386.801,E2 -7386.801} C_VEL
LIN {X 0,Y 474.92,Z 855.837,A -85,B 0,C 180,E1 -7387.868,E2 -7387.868} C_VEL
LIN {X 0,Y 475.167,Z 849.789,A -85,B 0,C 180,E1 -7388.934,E2 -7388.934} C_VEL
LIN {X 0,Y 475.427,Z 842.488,A -85,B 0,C 180,E1 -7390.003,E2 -7390.003} C_VEL
LIN {X 0,Y 475.683,Z 835.596,A -85,B 0,C 180,E1 -7390.858,E2 -7390.858} C_VEL
LIN {X 0,Y 476.015,Z 826.241,A -85,B 0,C 180,E1 -7391.821,E2 -7391.821} C_VEL
LIN {X 0,Y 476.289,Z 817.502,A -85,B 0,C 180,E1 -7392.571,E2 -7392.571} C_VEL
LIN {X 0,Y 476.554,Z 807.858,A -85,B 0,C 180,E1 -7393.253,E2 -7393.253} C_VEL
LIN {X 0,Y 476.83,Z 797.134,A -85,B 0,C 180,E1 -7393.858,E2 -7393.858} C_VEL
LIN {X 0,Y 477.024,Z 786.727,A -85,B 0,C 180,E1 -7394.314,E2 -7394.314} C_VEL
LIN {X 0,Y 477.127,Z 775.878,A -85,B 0,C 180,E1 -7394.665,E2 -7394.665} C_VEL
LIN {X 0,Y 477.252,Z 763.202,A -85,B 0,C 180,E1 -7394.934,E2 -7394.934} C_VEL
LIN {X 0,Y 477.737,Z 702.496,A -85,B 0,C 180,E1 -7395.923,E2 -7395.923} C_VEL
LIN {X 0,Y 474.676,Z 693.358,A -85,B 0,C 180,E1 -7396.179,E2 -7396.179} C_VEL
LIN {X 0,Y 474.675,Z 693.358,A -85,B 0,C 180,E1 -7399.01,E2 -7399.01} C_VEL
LIN {X 0,Y 474.601,Z 693.361,A -85,B 0,C 180,E1 -7401.728,E2 -7401.728} C_VEL
LIN {X 0,Y 474.643,Z 693.361,A -85,B 0,C 180,E1 -7404.494,E2 -7404.494} C_VEL
LIN {X 0,Y 474.653,Z 693.357,A -85,B 0,C 180,E1 -7407.323,E2 -7407.323} C_VEL
LIN {X 0,Y 474.616,Z 693.361,A -85,B 0,C 180,E1 -7410.23,E2 -7410.23} C_VEL
LIN {X 0,Y 474.63,Z 693.362,A -85,B 0,C 180,E1 -7413.221,E2 -7413.221} C_VEL
LIN {X 0,Y 474.599,Z 693.362,A -85,B 0,C 180,E1 -7416.323,E2 -7416.323} C_VEL
LIN {X 0,Y 474.637,Z 693.358,A -85,B 0,C 180,E1 -7419.547,E2 -7419.547} C_VEL
LIN {X 0,Y 474.601,Z 693.36,A -85,B 0,C 180,E1 -7422.23,E2 -7422.23} C_VEL
LIN {X 0,Y 474.63,Z 693.361,A -85,B 0,C 180,E1 -7425.296,E2 -7425.296} C_VEL
LIN {X 0,Y 474.607,Z 693.359,A -85,B 0,C 180,E1 -7428.209,E2 -7428.209} C_VEL
LIN {X 0,Y 474.632,Z 693.357,A -85,B 0,C 180,E1 -7430.449,E2 -7430.449} C_VEL
LIN {X 0,Y 474.583,Z 693.364,A -85,B 0,C 180,E1 -7433.672,E2 -7433.672} C_VEL
LIN {X 0,Y 474.623,Z 693.36,A -85,B 0,C 180,E1 -7436.774,E2 -7436.774} C_VEL
LIN {X 0,Y 474.564,Z 693.367,A -85,B 0,C 180,E1 -7439.763,E2 -7439.763} C_VEL
LIN {X 0,Y 474.584,Z 693.365,A -85,B 0,C 180,E1 -7440.772,E2 -7440.772} C_VEL
LIN {X 0,Y 473.944,Z 693.45,A -85,B 0,C 180,E1 -7441.481,E2 -7441.481} C_VEL
LIN {X 0,Y 471.128,Z 693.799,A -85,B 0,C 180,E1 -7442.632,E2 -7442.632} C_VEL
LIN {X 0,Y 468.719,Z 694.099,A -85,B 0,C 180,E1 -7443.56,E2 -7443.56} C_VEL
LIN {X 0,Y 467.66,Z 694.227,A -85,B 0,C 180,E1 -7444.277,E2 -7444.277} C_VEL
LIN {X 0,Y 467.561,Z 694.24,A -85,B 0,C 180,E1 -7444.52,E2 -7444.52} C_VEL
LIN {X 0,Y 467.564,Z 694.244,A -85,B 0,C 180,E1 -7446.991,E2 -7446.991} C_VEL
LIN {X 0,Y 467.548,Z 694.246,A -85,B 0,C 180,E1 -7449.769,E2 -7449.769} C_VEL
LIN {X 0,Y 467.58,Z 694.241,A -85,B 0,C 180,E1 -7452.501,E2 -7452.501} C_VEL
LIN {X 0,Y 467.574,Z 694.246,A -85,B 0,C 180,E1 -7453.401,E2 -7453.401} C_VEL
LIN {X 0,Y 471.39,Z 705.058,A -85,B 0,C 180,E1 -7453.724,E2 -7453.724} C_VEL
LIN {X 0,Y 470.965,Z 775.592,A -85,B 0,C 180,E1 -7454.83,E2 -7454.83} C_VEL
LIN {X 0,Y 470.989,Z 788.702,A -85,B 0,C 180,E1 -7455.217,E2 -7455.217} C_VEL
LIN {X 0,Y 470.778,Z 800.728,A -85,B 0,C 180,E1 -7455.736,E2 -7455.736} C_VEL
LIN {X 0,Y 470.485,Z 812.3,A -85,B 0,C 180,E1 -7456.406,E2 -7456.406} C_VEL
LIN {X 0,Y 470.036,Z 823.595,A -85,B 0,C 180,E1 -7457.254,E2 -7457.254} C_VEL
LIN {X 0,Y 469.621,Z 833.942,A -85,B 0,C 180,E1 -7458.23,E2 -7458.23} C_VEL
LIN {X 0,Y 469.25,Z 842.378,A -85,B 0,C 180,E1 -7459.205,E2 -7459.205} C_VEL
LIN {X 0,Y 468.834,Z 850.144,A -85,B 0,C 180,E1 -7460.286,E2 -7460.286} C_VEL
LIN {X 0,Y 468.381,Z 857.841,A -85,B 0,C 180,E1 -7461.604,E2 -7461.604} C_VEL
LIN {X 0,Y 468.208,Z 863.489,A -85,B 0,C 180,E1 -7462.812,E2 -7462.812} C_VEL
LIN {X 0,Y 467.88,Z 869.269,A -85,B 0,C 180,E1 -7464.392,E2 -7464.392} C_VEL
LIN {X 0,Y 467.607,Z 872.811,A -85,B 0,C 180,E1 -7465.685,E2 -7465.685} C_VEL
LIN {X 0,Y 467.499,Z 874.637,A -85,B 0,C 180,E1 -7466.547,E2 -7466.547} C_VEL
LIN {X 0,Y 467.498,Z 876.006,A -85,B 0,C 180,E1 -7467.41,E2 -7467.41} C_VEL
LIN {X 0,Y 467.448,Z 877.585,A -85,B 0,C 180,E1 -7469.133,E2 -7469.133} C_VEL
LIN {X 0,Y 467.428,Z 877.82,A -85,B 0,C 180,E1 -7469.994,E2 -7469.994} C_VEL
LIN {X 0,Y 467.536,Z 877.066,A -85,B 0,C 180,E1 -7471.717,E2 -7471.717} C_VEL
LIN {X 0,Y 467.49,Z 874.829,A -85,B 0,C 180,E1 -7473.442,E2 -7473.442} C_VEL
LIN {X 0,Y 467.675,Z 872.025,A -85,B 0,C 180,E1 -7474.735,E2 -7474.735} C_VEL
LIN {X 0,Y 467.942,Z 868.216,A -85,B 0,C 180,E1 -7476.029,E2 -7476.029} C_VEL
LIN {X 0,Y 468.173,Z 862.744,A -85,B 0,C 180,E1 -7477.459,E2 -7477.459} C_VEL
LIN {X 0,Y 468.521,Z 855.941,A -85,B 0,C 180,E1 -7478.838,E2 -7478.838} C_VEL
LIN {X 0,Y 468.977,Z 847.929,A -85,B 0,C 180,E1 -7480.135,E2 -7480.135} C_VEL
LIN {X 0,Y 469.404,Z 839.717,A -85,B 0,C 180,E1 -7481.217,E2 -7481.217} C_VEL
LIN {X 0,Y 469.8,Z 829.569,A -85,B 0,C 180,E1 -7482.302,E2 -7482.302} C_VEL
LIN {X 0,Y 470.305,Z 819.121,A -85,B 0,C 180,E1 -7483.194,E2 -7483.194} C_VEL
LIN {X 0,Y 470.651,Z 807.359,A -85,B 0,C 180,E1 -7483.994,E2 -7483.994} C_VEL
LIN {X 0,Y 470.865,Z 794.872,A -85,B 0,C 180,E1 -7484.631,E2 -7484.631} C_VEL
LIN {X 0,Y 471.036,Z 781.782,A -85,B 0,C 180,E1 -7485.101,E2 -7485.101} C_VEL
LIN {X 0,Y 471.031,Z 769.436,A -85,B 0,C 180,E1 -7485.378,E2 -7485.378} C_VEL
LIN {X 0,Y 471.456,Z 705.074,A -85,B 0,C 180,E1 -7486.366,E2 -7486.366} C_VEL
LIN {X 0,Y 467.59,Z 694.246,A -85,B 0,C 180,E1 -7486.687,E2 -7486.687} C_VEL
LIN {X 0,Y 467.606,Z 694.24,A -85,B 0,C 180,E1 -7489.301,E2 -7489.301} C_VEL
LIN {X 0,Y 467.514,Z 694.244,A -85,B 0,C 180,E1 -7492.067,E2 -7492.067} C_VEL
LIN {X 0,Y 467.547,Z 694.244,A -85,B 0,C 180,E1 -7494.882,E2 -7494.882} C_VEL
LIN {X 0,Y 467.589,Z 694.235,A -85,B 0,C 180,E1 -7497.762,E2 -7497.762} C_VEL
LIN {X 0,Y 467.537,Z 694.247,A -85,B 0,C 180,E1 -7501.038,E2 -7501.038} C_VEL
LIN {X 0,Y 467.555,Z 694.239,A -85,B 0,C 180,E1 -7504.236,E2 -7504.236} C_VEL
LIN {X 0,Y 467.511,Z 694.251,A -85,B 0,C 180,E1 -7507.18,E2 -7507.18} C_VEL
LIN {X 0,Y 467.555,Z 694.242,A -85,B 0,C 180,E1 -7510.256,E2 -7510.256} C_VEL
LIN {X 0,Y 467.575,Z 694.238,A -85,B 0,C 180,E1 -7512.565,E2 -7512.565} C_VEL
LIN {X 0,Y 467.525,Z 694.243,A -85,B 0,C 180,E1 -7516.17,E2 -7516.17} C_VEL
LIN {X 0,Y 467.539,Z 694.243,A -85,B 0,C 180,E1 -7518.715,E2 -7518.715} C_VEL
LIN {X 0,Y 467.527,Z 694.244,A -85,B 0,C 180,E1 -7521.4,E2 -7521.4} C_VEL
LIN {X 0,Y 467.505,Z 694.249,A -85,B 0,C 180,E1 -7524.255,E2 -7524.255} C_VEL
LIN {X 0,Y 467.522,Z 694.243,A -85,B 0,C 180,E1 -7527.316,E2 -7527.316} C_VEL
LIN {X 0,Y 467.514,Z 694.242,A -85,B 0,C 180,E1 -7530.661,E2 -7530.661} C_VEL
LIN {X 0,Y 467.561,Z 694.238,A -85,B 0,C 180,E1 -7533.196,E2 -7533.196} C_VEL
LIN {X 0,Y 467.507,Z 694.249,A -85,B 0,C 180,E1 -7536.053,E2 -7536.053} C_VEL
LIN {X 0,Y 467.552,Z 694.241,A -85,B 0,C 180,E1 -7539.774,E2 -7539.774} C_VEL
LIN {X 0,Y 467.538,Z 694.243,A -85,B 0,C 180,E1 -7542.504,E2 -7542.504} C_VEL
LIN {X 0,Y 467.543,Z 694.243,A -85,B 0,C 180,E1 -7545.194,E2 -7545.194} C_VEL
LIN {X 0,Y 467.623,Z 694.23,A -85,B 0,C 180,E1 -7547.854,E2 -7547.854} C_VEL
LIN {X 0,Y 467.613,Z 694.234,A -85,B 0,C 180,E1 -7551.356,E2 -7551.356} C_VEL
LIN {X 0,Y 467.678,Z 694.225,A -85,B 0,C 180,E1 -7553.962,E2 -7553.962} C_VEL
LIN {X 0,Y 467.792,Z 694.213,A -85,B 0,C 180,E1 -7557.417,E2 -7557.417} C_VEL
LIN {X 0,Y 467.803,Z 694.211,A -85,B 0,C 180,E1 -7560,E2 -7560} C_VEL
LIN {X 0,Y 467.792,Z 694.21,A -85,B 0,C 180,E1 -7562.583,E2 -7562.583} C_VEL
LIN {X 0,Y 467.678,Z 694.226,A -85,B 0,C 180,E1 -7566.038,E2 -7566.038} C_VEL
LIN {X 0,Y 467.613,Z 694.232,A -85,B 0,C 180,E1 -7568.644,E2 -7568.644} C_VEL
LIN {X 0,Y 467.623,Z 694.232,A -85,B 0,C 180,E1 -7572.146,E2 -7572.146} C_VEL
LIN {X 0,Y 467.594,Z 694.237,A -85,B 0,C 180,E1 -7575.896,E2 -7575.896} C_VEL
LIN {X 0,Y 467.552,Z 694.245,A -85,B 0,C 180,E1 -7579.311,E2 -7579.311} C_VEL
LIN {X 0,Y 467.472,Z 694.252,A -85,B 0,C 180,E1 -7582.077,E2 -7582.077} C_VEL
LIN {X 0,Y 467.553,Z 694.238,A -85,B 0,C 180,E1 -7584.89,E2 -7584.89} C_VEL
LIN {X 0,Y 467.563,Z 694.245,A -85,B 0,C 180,E1 -7587.773,E2 -7587.773} C_VEL
LIN {X 0,Y 467.513,Z 694.242,A -85,B 0,C 180,E1 -7591.051,E2 -7591.051} C_VEL
LIN {X 0,Y 467.53,Z 694.247,A -85,B 0,C 180,E1 -7594.248,E2 -7594.248} C_VEL
LIN {X 0,Y 467.495,Z 694.246,A -85,B 0,C 180,E1 -7597.192,E2 -7597.192} C_VEL
LIN {X 0,Y 467.549,Z 694.244,A -85,B 0,C 180,E1 -7600.268,E2 -7600.268} C_VEL
LIN {X 0,Y 467.569,Z 694.243,A -85,B 0,C 180,E1 -7602.577,E2 -7602.577} C_VEL
LIN {X 0,Y 467.53,Z 694.251,A -85,B 0,C 180,E1 -7606.264,E2 -7606.264} C_VEL
LIN {X 0,Y 467.547,Z 694.247,A -85,B 0,C 180,E1 -7608.728,E2 -7608.728} C_VEL
LIN {X 0,Y 467.534,Z 694.244,A -85,B 0,C 180,E1 -7611.414,E2 -7611.414} C_VEL
LIN {X 0,Y 467.525,Z 694.248,A -85,B 0,C 180,E1 -7614.267,E2 -7614.267} C_VEL
LIN {X 0,Y 467.549,Z 694.244,A -85,B 0,C 180,E1 -7617.328,E2 -7617.328} C_VEL
LIN {X 0,Y 467.585,Z 694.367,A -85,B 0,C 180,E1 -7619.433,E2 -7619.433} C_VEL
LIN {X 0,Y 471.572,Z 711.779,A -85,B 0,C 180,E1 -7622.065,E2 -7622.065} C_VEL
LIN {X 0,Y 471.629,Z 716.678,A -85,B 0,C 180,E1 -7622.736,E2 -7622.736} C_VEL
LIN {X 0,Y 470.717,Z 737.66,A -85,B 0,C 180,E1 -7625.521,E2 -7625.521} C_VEL
LIN {X 0,Y 469.758,Z 762.173,A -85,B 0,C 180,E1 -7628.735,E2 -7628.735} C_VEL
LIN {X 0,Y 468.814,Z 787.978,A -85,B 0,C 180,E1 -7632.11,E2 -7632.11} C_VEL
LIN {X 0,Y 468.608,Z 794.444,A -85,B 0,C 180,E1 -7632.957,E2 -7632.957} C_VEL
LIN {X 0,Y 471.085,Z 818.04,A -85,B 0,C 180,E1 -7633.418,E2 -7633.418} C_VEL
LIN {X 0,Y 470.383,Z 905.285,A -85,B 0,C 180,E1 -7634.767,E2 -7634.767} C_VEL
LIN {X 0,Y 469.963,Z 918.53,A -85,B 0,C 180,E1 -7635.141,E2 -7635.141} C_VEL
LIN {X 0,Y 469.5,Z 931.876,A -85,B 0,C 180,E1 -7635.707,E2 -7635.707} C_VEL
LIN {X 0,Y 469.032,Z 943.127,A -85,B 0,C 180,E1 -7636.356,E2 -7636.356} C_VEL
LIN {X 0,Y 468.516,Z 954.884,A -85,B 0,C 180,E1 -7637.226,E2 -7637.226} C_VEL
LIN {X 0,Y 468.082,Z 965.455,A -85,B 0,C 180,E1 -7638.202,E2 -7638.202} C_VEL
LIN {X 0,Y 467.721,Z 974.144,A -85,B 0,C 180,E1 -7639.181,E2 -7639.181} C_VEL
LIN {X 0,Y 467.396,Z 982.177,A -85,B 0,C 180,E1 -7640.267,E2 -7640.267} C_VEL
LIN {X 0,Y 467.147,Z 990.051,A -85,B 0,C 180,E1 -7641.572,E2 -7641.572} C_VEL
LIN {X 0,Y 466.966,Z 997.323,A -85,B 0,C 180,E1 -7643.091,E2 -7643.091} C_VEL
LIN {X 0,Y 466.918,Z 1002.178,A -85,B 0,C 180,E1 -7644.391,E2 -7644.391} C_VEL
LIN {X 0,Y 466.875,Z 1005.893,A -85,B 0,C 180,E1 -7645.69,E2 -7645.69} C_VEL
LIN {X 0,Y 466.895,Z 1007.815,A -85,B 0,C 180,E1 -7646.554,E2 -7646.554} C_VEL
LIN {X 0,Y 466.859,Z 1009.247,A -85,B 0,C 180,E1 -7647.417,E2 -7647.417} C_VEL
LIN {X 0,Y 466.846,Z 1010.27,A -85,B 0,C 180,E1 -7648.28,E2 -7648.28} C_VEL
LIN {X 0,Y 466.822,Z 1010.891,A -85,B 0,C 180,E1 -7649.143,E2 -7649.143} C_VEL
LIN {X 0,Y 466.82,Z 1011.11,A -85,B 0,C 180,E1 -7650.006,E2 -7650.006} C_VEL
LIN {X 0,Y 466.822,Z 1010.884,A -85,B 0,C 180,E1 -7650.868,E2 -7650.868} C_VEL
LIN {X 0,Y 466.847,Z 1010.258,A -85,B 0,C 180,E1 -7651.731,E2 -7651.731} C_VEL
LIN {X 0,Y 466.861,Z 1009.229,A -85,B 0,C 180,E1 -7652.594,E2 -7652.594} C_VEL
LIN {X 0,Y 466.898,Z 1007.79,A -85,B 0,C 180,E1 -7653.457,E2 -7653.457} C_VEL
LIN {X 0,Y 466.892,Z 1004.76,A -85,B 0,C 180,E1 -7654.754,E2 -7654.754} C_VEL
LIN {X 0,Y 466.951,Z 999.664,A -85,B 0,C 180,E1 -7656.321,E2 -7656.321} C_VEL
LIN {X 0,Y 467.049,Z 993.339,A -85,B 0,C 180,E1 -7657.789,E2 -7657.789} C_VEL
LIN {X 0,Y 467.264,Z 986.266,A -85,B 0,C 180,E1 -7659.092,E2 -7659.092} C_VEL
LIN {X 0,Y 467.543,Z 977.426,A -85,B 0,C 180,E1 -7660.397,E2 -7660.397} C_VEL
LIN {X 0,Y 467.96,Z 968.406,A -85,B 0,C 180,E1 -7661.483,E2 -7661.483} C_VEL
LIN {X 0,Y 468.399,Z 958.5,A -85,B 0,C 180,E1 -7662.463,E2 -7662.463} C_VEL
LIN {X 0,Y 468.87,Z 947.734,A -85,B 0,C 180,E1 -7663.329,E2 -7663.329} C_VEL
LIN {X 0,Y 469.335,Z 935.706,A -85,B 0,C 180,E1 -7664.088,E2 -7664.088} C_VEL
LIN {X 0,Y 469.813,Z 923.237,A -85,B 0,C 180,E1 -7664.682,E2 -7664.682} C_VEL
LIN {X 0,Y 470.254,Z 910.443,A -85,B 0,C 180,E1 -7665.111,E2 -7665.111} C_VEL
LIN {X 0,Y 470.481,Z 897.007,A -85,B 0,C 180,E1 -7665.381,E2 -7665.381} C_VEL
LIN {X 0,Y 471.088,Z 816.428,A -85,B 0,C 180,E1 -7666.607,E2 -7666.607} C_VEL
LIN {X 0,Y 468.579,Z 794.467,A -85,B 0,C 180,E1 -7667.039,E2 -7667.039} C_VEL
LIN {X 0,Y 469.431,Z 770.729,A -85,B 0,C 180,E1 -7670.146,E2 -7670.146} C_VEL
LIN {X 0,Y 470.373,Z 746.378,A -85,B 0,C 180,E1 -7673.329,E2 -7673.329} C_VEL
LIN {X 0,Y 471.28,Z 724.155,A -85,B 0,C 180,E1 -7676.265,E2 -7676.265} C_VEL
LIN {X 0,Y 471.772,Z 713.308,A -85,B 0,C 180,E1 -7677.715,E2 -7677.715} C_VEL
LIN {X 0,Y 468.101,Z 696.744,A -85,B 0,C 180,E1 -7680.201,E2 -7680.201} C_VEL
LIN {X 0,Y 467.575,Z 694.243,A -85,B 0,C 180,E1 -7680.613,E2 -7680.613} C_VEL
LIN {X 0,Y 467.523,Z 694.25,A -85,B 0,C 180,E1 -7683.798,E2 -7683.798} C_VEL
LIN {X 0,Y 467.514,Z 694.25,A -85,B 0,C 180,E1 -7687.18,E2 -7687.18} C_VEL
LIN {X 0,Y 467.532,Z 694.244,A -85,B 0,C 180,E1 -7690.273,E2 -7690.273} C_VEL
LIN {X 0,Y 467.532,Z 694.244,A -85,B 0,C 180,E1 -7692.571,E2 -7692.571} C_VEL
LIN {X 0,Y 467.57,Z 694.243,A -85,B 0,C 180,E1 -7695.053,E2 -7695.053} C_VEL
LIN {X 0,Y 467.576,Z 694.24,A -85,B 0,C 180,E1 -7698.728,E2 -7698.728} C_VEL
LIN {X 0,Y 467.558,Z 694.241,A -85,B 0,C 180,E1 -7701.955,E2 -7701.955} C_VEL
LIN {X 0,Y 467.569,Z 694.244,A -85,B 0,C 180,E1 -7705.168,E2 -7705.168} C_VEL
LIN {X 0,Y 467.596,Z 694.235,A -85,B 0,C 180,E1 -7708.261,E2 -7708.261} C_VEL
LIN {X 0,Y 467.563,Z 694.246,A -85,B 0,C 180,E1 -7711.249,E2 -7711.249} C_VEL
LIN {X 0,Y 467.607,Z 694.236,A -85,B 0,C 180,E1 -7714.398,E2 -7714.398} C_VEL
LIN {X 0,Y 467.587,Z 694.242,A -85,B 0,C 180,E1 -7716.996,E2 -7716.996} C_VEL
LIN {X 0,Y 467.636,Z 694.237,A -85,B 0,C 180,E1 -7719.778,E2 -7719.778} C_VEL
LIN {X 0,Y 467.61,Z 694.237,A -85,B 0,C 180,E1 -7722.507,E2 -7722.507} C_VEL
LIN {X 0,Y 467.61,Z 694.241,A -85,B 0,C 180,E1 -7723.531,E2 -7723.531} C_VEL
LIN {X 0,Y 471.073,Z 703.881,A -85,B 0,C 180,E1 -7723.862,E2 -7723.862} C_VEL
LIN {X 0,Y 470.36,Z 774.844,A -85,B 0,C 180,E1 -7725.119,E2 -7725.119} C_VEL
LIN {X 0,Y 470.291,Z 787.112,A -85,B 0,C 180,E1 -7725.476,E2 -7725.476} C_VEL
LIN {X 0,Y 470.197,Z 797.127,A -85,B 0,C 180,E1 -7725.888,E2 -7725.888} C_VEL
LIN {X 0,Y 469.942,Z 807.456,A -85,B 0,C 180,E1 -7726.436,E2 -7726.436} C_VEL
LIN {X 0,Y 469.701,Z 816.443,A -85,B 0,C 180,E1 -7727.03,E2 -7727.03} C_VEL
LIN {X 0,Y 469.379,Z 825.828,A -85,B 0,C 180,E1 -7727.79,E2 -7727.79} C_VEL
LIN {X 0,Y 469.114,Z 833.671,A -85,B 0,C 180,E1 -7728.551,E2 -7728.551} C_VEL
LIN {X 0,Y 468.838,Z 841.221,A -85,B 0,C 180,E1 -7729.419,E2 -7729.419} C_VEL
LIN {X 0,Y 468.474,Z 849.021,A -85,B 0,C 180,E1 -7730.502,E2 -7730.502} C_VEL
LIN {X 0,Y 468.217,Z 855.469,A -85,B 0,C 180,E1 -7731.585,E2 -7731.585} C_VEL
LIN {X 0,Y 467.989,Z 861.161,A -85,B 0,C 180,E1 -7732.748,E2 -7732.748} C_VEL
LIN {X 0,Y 467.791,Z 865.949,A -85,B 0,C 180,E1 -7733.963,E2 -7733.963} C_VEL
LIN {X 0,Y 467.56,Z 868.814,A -85,B 0,C 180,E1 -7734.826,E2 -7734.826} C_VEL
LIN {X 0,Y 467.403,Z 872.812,A -85,B 0,C 180,E1 -7736.552,E2 -7736.552} C_VEL
LIN {X 0,Y 467.411,Z 874.268,A -85,B 0,C 180,E1 -7737.415,E2 -7737.415} C_VEL
LIN {X 0,Y 467.352,Z 875.752,A -85,B 0,C 180,E1 -7739.138,E2 -7739.138} C_VEL
LIN {X 0,Y 467.32,Z 875.915,A -85,B 0,C 180,E1 -7740,E2 -7740} C_VEL
LIN {X 0,Y 467.31,Z 875.642,A -85,B 0,C 180,E1 -7740.862,E2 -7740.862} C_VEL
LIN {X 0,Y 467.221,Z 873.9,A -85,B 0,C 180,E1 -7742.586,E2 -7742.586} C_VEL
LIN {X 0,Y 467.401,Z 870.412,A -85,B 0,C 180,E1 -7744.312,E2 -7744.312} C_VEL
LIN {X 0,Y 467.532,Z 866.637,A -85,B 0,C 180,E1 -7745.607,E2 -7745.607} C_VEL
LIN {X 0,Y 467.805,Z 861.705,A -85,B 0,C 180,E1 -7746.903,E2 -7746.903} C_VEL
LIN {X 0,Y 467.953,Z 856.66,A -85,B 0,C 180,E1 -7747.986,E2 -7747.986} C_VEL
LIN {X 0,Y 468.218,Z 850.561,A -85,B 0,C 180,E1 -7749.068,E2 -7749.068} C_VEL
LIN {X 0,Y 468.481,Z 843.198,A -85,B 0,C 180,E1 -7750.153,E2 -7750.153} C_VEL
LIN {X 0,Y 468.763,Z 836.245,A -85,B 0,C 180,E1 -7751.02,E2 -7751.02} C_VEL
LIN {X 0,Y 469.093,Z 826.807,A -85,B 0,C 180,E1 -7751.998,E2 -7751.998} C_VEL
LIN {X 0,Y 469.378,Z 817.975,A -85,B 0,C 180,E1 -7752.759,E2 -7752.759} C_VEL
LIN {X 0,Y 469.669,Z 808.622,A -85,B 0,C 180,E1 -7753.426,E2 -7753.426} C_VEL
LIN {X 0,Y 469.92,Z 798.457,A -85,B 0,C 180,E1 -7754.01,E2 -7754.01} C_VEL
LIN {X 0,Y 470.13,Z 788.18,A -85,B 0,C 180,E1 -7754.473,E2 -7754.473} C_VEL
LIN {X 0,Y 470.224,Z 777.585,A -85,B 0,C 180,E1 -7754.83,E2 -7754.83} C_VEL
LIN {X 0,Y 470.342,Z 765.384,A -85,B 0,C 180,E1 -7755.103,E2 -7755.103} C_VEL
LIN {X 0,Y 470.763,Z 703.693,A -85,B 0,C 180,E1 -7756.134,E2 -7756.134} C_VEL
LIN {X 0,Y 467.612,Z 694.24,A -85,B 0,C 180,E1 -7756.409,E2 -7756.409} C_VEL
LIN {X 0,Y 467.635,Z 694.232,A -85,B 0,C 180,E1 -7759.307,E2 -7759.307} C_VEL
LIN {X 0,Y 467.545,Z 694.241,A -85,B 0,C 180,E1 -7762.073,E2 -7762.073} C_VEL
LIN {X 0,Y 467.584,Z 694.243,A -85,B 0,C 180,E1 -7764.889,E2 -7764.889} C_VEL
LIN {X 0,Y 467.595,Z 694.233,A -85,B 0,C 180,E1 -7767.771,E2 -7767.771} C_VEL
LIN {X 0,Y 467.582,Z 694.243,A -85,B 0,C 180,E1 -7771.043,E2 -7771.043} C_VEL
LIN {X 0,Y 467.592,Z 694.235,A -85,B 0,C 180,E1 -7774.238,E2 -7774.238} C_VEL
LIN {X 0,Y 467.558,Z 694.244,A -85,B 0,C 180,E1 -7777.184,E2 -7777.184} C_VEL
LIN {X 0,Y 467.574,Z 694.237,A -85,B 0,C 180,E1 -7780.265,E2 -7780.265} C_VEL
LIN {X 0,Y 467.562,Z 694.237,A -85,B 0,C 180,E1 -7783.744,E2 -7783.744} C_VEL
LIN {X 0,Y 467.546,Z 694.239,A -85,B 0,C 180,E1 -7786.25,E2 -7786.25} C_VEL
LIN {X 0,Y 467.577,Z 694.238,A -85,B 0,C 180,E1 -7788.724,E2 -7788.724} C_VEL
LIN {X 0,Y 467.554,Z 694.238,A -85,B 0,C 180,E1 -7791.95,E2 -7791.95} C_VEL
LIN {X 0,Y 467.557,Z 694.244,A -85,B 0,C 180,E1 -7795.163,E2 -7795.163} C_VEL
LIN {X 0,Y 467.558,Z 694.238,A -85,B 0,C 180,E1 -7798.254,E2 -7798.254} C_VEL
LIN {X 0,Y 467.535,Z 694.248,A -85,B 0,C 180,E1 -7801.243,E2 -7801.243} C_VEL
LIN {X 0,Y 467.561,Z 694.24,A -85,B 0,C 180,E1 -7804.52,E2 -7804.52} C_VEL
LIN {X 0,Y 466.855,Z 694.333,A -85,B 0,C 180,E1 -7805.238,E2 -7805.238} C_VEL
LIN {X 0,Y 463.975,Z 694.69,A -85,B 0,C 180,E1 -7806.406,E2 -7806.406} C_VEL
LIN {X 0,Y 461.578,Z 694.992,A -85,B 0,C 180,E1 -7807.347,E2 -7807.347} C_VEL
LIN {X 0,Y 460.576,Z 695.112,A -85,B 0,C 180,E1 -7808.074,E2 -7808.074} C_VEL
LIN {X 0,Y 460.507,Z 695.12,A -85,B 0,C 180,E1 -7808.32,E2 -7808.32} C_VEL
LIN {X 0,Y 460.539,Z 695.122,A -85,B 0,C 180,E1 -7811.304,E2 -7811.304} C_VEL
LIN {X 0,Y 460.546,Z 695.121,A -85,B 0,C 180,E1 -7813.141,E2 -7813.141} C_VEL
LIN {X 0,Y 464.668,Z 706.642,A -85,B 0,C 180,E1 -7813.49,E2 -7813.49} C_VEL
LIN {X 0,Y 464.189,Z 776.612,A -85,B 0,C 180,E1 -7814.603,E2 -7814.603} C_VEL
LIN {X 0,Y 464.196,Z 789.716,A -85,B 0,C 180,E1 -7814.996,E2 -7814.996} C_VEL
LIN {X 0,Y 463.968,Z 801.74,A -85,B 0,C 180,E1 -7815.522,E2 -7815.522} C_VEL
LIN {X 0,Y 463.657,Z 813.304,A -85,B 0,C 180,E1 -7816.202,E2 -7816.202} C_VEL
LIN {X 0,Y 463.185,Z 824.603,A -85,B 0,C 180,E1 -7817.062,E2 -7817.062} C_VEL
LIN {X 0,Y 462.745,Z 834.949,A -85,B 0,C 180,E1 -7818.052,E2 -7818.052} C_VEL
LIN {X 0,Y 462.352,Z 843.384,A -85,B 0,C 180,E1 -7819.042,E2 -7819.042} C_VEL
LIN {X 0,Y 461.911,Z 851.149,A -85,B 0,C 180,E1 -7820.139,E2 -7820.139} C_VEL
LIN {X 0,Y 461.457,Z 858.842,A -85,B 0,C 180,E1 -7821.477,E2 -7821.477} C_VEL
LIN {X 0,Y 461.237,Z 864.493,A -85,B 0,C 180,E1 -7822.703,E2 -7822.703} C_VEL
LIN {X 0,Y 460.912,Z 870.269,A -85,B 0,C 180,E1 -7824.307,E2 -7824.307} C_VEL
LIN {X 0,Y 460.598,Z 873.815,A -85,B 0,C 180,E1 -7825.619,E2 -7825.619} C_VEL
LIN {X 0,Y 460.483,Z 875.641,A -85,B 0,C 180,E1 -7826.494,E2 -7826.494} C_VEL
LIN {X 0,Y 460.482,Z 877.008,A -85,B 0,C 180,E1 -7827.37,E2 -7827.37} C_VEL
LIN {X 0,Y 460.428,Z 878.587,A -85,B 0,C 180,E1 -7829.12,E2 -7829.12} C_VEL
LIN {X 0,Y 460.407,Z 878.822,A -85,B 0,C 180,E1 -7829.994,E2 -7829.994} C_VEL
LIN {X 0,Y 460.52,Z 878.067,A -85,B 0,C 180,E1 -7831.743,E2 -7831.743} C_VEL
LIN {X 0,Y 460.474,Z 875.832,A -85,B 0,C 180,E1 -7833.494,E2 -7833.494} C_VEL
LIN {X 0,Y 460.671,Z 873.027,A -85,B 0,C 180,E1 -7834.807,E2 -7834.807} C_VEL
LIN {X 0,Y 460.96,Z 869.216,A -85,B 0,C 180,E1 -7836.12,E2 -7836.12} C_VEL
LIN {X 0,Y 461.206,Z 863.744,A -85,B 0,C 180,E1 -7837.572,E2 -7837.572} C_VEL
LIN {X 0,Y 461.579,Z 856.941,A -85,B 0,C 180,E1 -7838.972,E2 -7838.972} C_VEL
LIN {X 0,Y 462.063,Z 848.928,A -85,B 0,C 180,E1 -7840.288,E2 -7840.288} C_VEL
LIN {X 0,Y 462.515,Z 840.716,A -85,B 0,C 180,E1 -7841.386,E2 -7841.386} C_VEL
LIN {X 0,Y 462.936,Z 830.567,A -85,B 0,C 180,E1 -7842.487,E2 -7842.487} C_VEL
LIN {X 0,Y 463.466,Z 820.118,A -85,B 0,C 180,E1 -7843.393,E2 -7843.393} C_VEL
LIN {X 0,Y 463.834,Z 808.355,A -85,B 0,C 180,E1 -7844.204,E2 -7844.204} C_VEL
LIN {X 0,Y 464.059,Z 795.866,A -85,B 0,C 180,E1 -7844.851,E2 -7844.851} C_VEL
LIN {X 0,Y 464.232,Z 782.773,A -85,B 0,C 180,E1 -7845.328,E2 -7845.328} C_VEL
LIN {X 0,Y 464.236,Z 770.414,A -85,B 0,C 180,E1 -7845.609,E2 -7845.609} C_VEL
LIN {X 0,Y 464.632,Z 706.493,A -85,B 0,C 180,E1 -7846.607,E2 -7846.607} C_VEL
LIN {X 0,Y 460.554,Z 695.131,A -85,B 0,C 180,E1 -7846.95,E2 -7846.95} C_VEL
LIN {X 0,Y 460.552,Z 695.116,A -85,B 0,C 180,E1 -7849.609,E2 -7849.609} C_VEL
LIN {X 0,Y 460.49,Z 695.12,A -85,B 0,C 180,E1 -7852.422,E2 -7852.422} C_VEL
LIN {X 0,Y 460.522,Z 695.114,A -85,B 0,C 180,E1 -7855.789,E2 -7855.789} C_VEL
LIN {X 0,Y 460.522,Z 695.114,A -85,B 0,C 180,E1 -7858.226,E2 -7858.226} C_VEL
LIN {X 0,Y 460.49,Z 695.127,A -85,B 0,C 180,E1 -7861.276,E2 -7861.276} C_VEL
LIN {X 0,Y 460.499,Z 695.118,A -85,B 0,C 180,E1 -7864.499,E2 -7864.499} C_VEL
LIN {X 0,Y 460.491,Z 695.117,A -85,B 0,C 180,E1 -7867.614,E2 -7867.614} C_VEL
LIN {X 0,Y 460.518,Z 695.118,A -85,B 0,C 180,E1 -7870.265,E2 -7870.265} C_VEL
LIN {X 0,Y 460.48,Z 695.127,A -85,B 0,C 180,E1 -7873.366,E2 -7873.366} C_VEL
LIN {X 0,Y 460.475,Z 695.118,A -85,B 0,C 180,E1 -7876.621,E2 -7876.621} C_VEL
LIN {X 0,Y 460.512,Z 695.126,A -85,B 0,C 180,E1 -7879.721,E2 -7879.721} C_VEL
LIN {X 0,Y 460.473,Z 695.123,A -85,B 0,C 180,E1 -7882.513,E2 -7882.513} C_VEL
LIN {X 0,Y 460.489,Z 695.122,A -85,B 0,C 180,E1 -7885.619,E2 -7885.619} C_VEL
LIN {X 0,Y 460.475,Z 695.122,A -85,B 0,C 180,E1 -7888.74,E2 -7888.74} C_VEL
LIN {X 0,Y 460.493,Z 695.117,A -85,B 0,C 180,E1 -7891.763,E2 -7891.763} C_VEL
LIN {X 0,Y 460.515,Z 695.117,A -85,B 0,C 180,E1 -7894.703,E2 -7894.703} C_VEL
LIN {X 0,Y 460.444,Z 695.123,A -85,B 0,C 180,E1 -7897.568,E2 -7897.568} C_VEL
LIN {X 0,Y 460.498,Z 695.126,A -85,B 0,C 180,E1 -7900.381,E2 -7900.381} C_VEL
LIN {X 0,Y 460.558,Z 695.11,A -85,B 0,C 180,E1 -7904.057,E2 -7904.057} C_VEL
LIN {X 0,Y 460.583,Z 695.107,A -85,B 0,C 180,E1 -7907.665,E2 -7907.665} C_VEL
LIN {X 0,Y 460.56,Z 695.114,A -85,B 0,C 180,E1 -7911.222,E2 -7911.222} C_VEL
LIN {X 0,Y 460.642,Z 695.102,A -85,B 0,C 180,E1 -7913.869,E2 -7913.869} C_VEL
LIN {X 0,Y 460.758,Z 695.089,A -85,B 0,C 180,E1 -7917.377,E2 -7917.377} C_VEL
LIN {X 0,Y 460.774,Z 695.086,A -85,B 0,C 180,E1 -7920,E2 -7920} C_VEL
LIN {X 0,Y 460.758,Z 695.086,A -85,B 0,C 180,E1 -7922.623,E2 -7922.623} C_VEL
LIN {X 0,Y 460.642,Z 695.103,A -85,B 0,C 180,E1 -7926.131,E2 -7926.131} C_VEL
LIN {X 0,Y 460.56,Z 695.112,A -85,B 0,C 180,E1 -7928.777,E2 -7928.777} C_VEL
LIN {X 0,Y 460.583,Z 695.109,A -85,B 0,C 180,E1 -7932.335,E2 -7932.335} C_VEL
LIN {X 0,Y 460.549,Z 695.113,A -85,B 0,C 180,E1 -7936.01,E2 -7936.01} C_VEL
LIN {X 0,Y 460.498,Z 695.122,A -85,B 0,C 180,E1 -7939.619,E2 -7939.619} C_VEL
LIN {X 0,Y 460.446,Z 695.125,A -85,B 0,C 180,E1 -7942.432,E2 -7942.432} C_VEL
LIN {X 0,Y 460.519,Z 695.118,A -85,B 0,C 180,E1 -7945.811,E2 -7945.811} C_VEL
LIN {X 0,Y 460.493,Z 695.122,A -85,B 0,C 180,E1 -7948.237,E2 -7948.237} C_VEL
LIN {X 0,Y 460.465,Z 695.122,A -85,B 0,C 180,E1 -7951.289,E2 -7951.289} C_VEL
LIN {X 0,Y 460.474,Z 695.124,A -85,B 0,C 180,E1 -7954.511,E2 -7954.511} C_VEL
LIN {X 0,Y 460.475,Z 695.123,A -85,B 0,C 180,E1 -7957.626,E2 -7957.626} C_VEL
LIN {X 0,Y 460.512,Z 695.12,A -85,B 0,C 180,E1 -7960.279,E2 -7960.279} C_VEL
LIN {X 0,Y 460.475,Z 695.122,A -85,B 0,C 180,E1 -7963.379,E2 -7963.379} C_VEL
LIN {X 0,Y 460.479,Z 695.123,A -85,B 0,C 180,E1 -7966.634,E2 -7966.634} C_VEL
LIN {X 0,Y 460.517,Z 695.119,A -85,B 0,C 180,E1 -7969.735,E2 -7969.735} C_VEL
LIN {X 0,Y 460.488,Z 695.127,A -85,B 0,C 180,E1 -7972.526,E2 -7972.526} C_VEL
LIN {X 0,Y 460.513,Z 695.115,A -85,B 0,C 180,E1 -7975.631,E2 -7975.631} C_VEL
LIN {X 0,Y 460.516,Z 695.124,A -85,B 0,C 180,E1 -7979.135,E2 -7979.135} C_VEL
LIN {X 0,Y 464.519,Z 712.674,A -85,B 0,C 180,E1 -7981.857,E2 -7981.857} C_VEL
LIN {X 0,Y 464.845,Z 715.778,A -85,B 0,C 180,E1 -7982.304,E2 -7982.304} C_VEL
LIN {X 0,Y 464.011,Z 733.305,A -85,B 0,C 180,E1 -7984.675,E2 -7984.675} C_VEL
LIN {X 0,Y 462.982,Z 757.649,A -85,B 0,C 180,E1 -7987.927,E2 -7987.927} C_VEL
LIN {X 0,Y 461.978,Z 783.585,A -85,B 0,C 180,E1 -7991.377,E2 -7991.377} C_VEL
LIN {X 0,Y 461.592,Z 793.343,A -85,B 0,C 180,E1 -7992.678,E2 -7992.678} C_VEL
LIN {X 0,Y 464.259,Z 817.031,A -85,B 0,C 180,E1 -7993.167,E2 -7993.167} C_VEL
LIN {X 0,Y 463.53,Z 904.274,A -85,B 0,C 180,E1 -7994.536,E2 -7994.536} C_VEL
LIN {X 0,Y 463.114,Z 917.52,A -85,B 0,C 180,E1 -7994.916,E2 -7994.916} C_VEL
LIN {X 0,Y 462.659,Z 929.734,A -85,B 0,C 180,E1 -7995.435,E2 -7995.435} C_VEL
LIN {X 0,Y 462.061,Z 942.104,A -85,B 0,C 180,E1 -7996.146,E2 -7996.146} C_VEL
LIN {X 0,Y 461.524,Z 954.158,A -85,B 0,C 180,E1 -7997.054,E2 -7997.054} C_VEL
LIN {X 0,Y 461.091,Z 964.435,A -85,B 0,C 180,E1 -7998.021,E2 -7998.021} C_VEL
LIN {X 0,Y 460.674,Z 973.12,A -85,B 0,C 180,E1 -7999.013,E2 -7999.013} C_VEL
LIN {X 0,Y 460.338,Z 981.155,A -85,B 0,C 180,E1 -8000.117,E2 -8000.117} C_VEL
LIN {X 0,Y 460.106,Z 989.036,A -85,B 0,C 180,E1 -8001.442,E2 -8001.442} C_VEL
LIN {X 0,Y 459.913,Z 996.309,A -85,B 0,C 180,E1 -8002.984,E2 -8002.984} C_VEL
LIN {X 0,Y 459.863,Z 1001.167,A -85,B 0,C 180,E1 -8004.305,E2 -8004.305} C_VEL
LIN {X 0,Y 459.83,Z 1004.885,A -85,B 0,C 180,E1 -8005.623,E2 -8005.623} C_VEL
LIN {X 0,Y 459.853,Z 1006.808,A -85,B 0,C 180,E1 -8006.501,E2 -8006.501} C_VEL
LIN {X 0,Y 459.819,Z 1008.242,A -85,B 0,C 180,E1 -8007.378,E2 -8007.378} C_VEL
LIN {X 0,Y 459.811,Z 1009.266,A -85,B 0,C 180,E1 -8008.254,E2 -8008.254} C_VEL
LIN {X 0,Y 459.792,Z 1009.888,A -85,B 0,C 180,E1 -8009.13,E2 -8009.13} C_VEL
LIN {X 0,Y 459.791,Z 1010.107,A -85,B 0,C 180,E1 -8010.006,E2 -8010.006} C_VEL
LIN {X 0,Y 459.792,Z 1009.881,A -85,B 0,C 180,E1 -8010.882,E2 -8010.882} C_VEL
LIN {X 0,Y 459.812,Z 1009.254,A -85,B 0,C 180,E1 -8011.757,E2 -8011.757} C_VEL
LIN {X 0,Y 459.82,Z 1008.224,A -85,B 0,C 180,E1 -8012.634,E2 -8012.634} C_VEL
LIN {X 0,Y 459.856,Z 1006.783,A -85,B 0,C 180,E1 -8013.51,E2 -8013.51} C_VEL
LIN {X 0,Y 459.849,Z 1003.752,A -85,B 0,C 180,E1 -8014.827,E2 -8014.827} C_VEL
LIN {X 0,Y 459.894,Z 999.659,A -85,B 0,C 180,E1 -8016.146,E2 -8016.146} C_VEL
LIN {X 0,Y 459.978,Z 993.362,A -85,B 0,C 180,E1 -8017.688,E2 -8017.688} C_VEL
LIN {X 0,Y 460.148,Z 986.508,A -85,B 0,C 180,E1 -8019.012,E2 -8019.012} C_VEL
LIN {X 0,Y 460.451,Z 978.034,A -85,B 0,C 180,E1 -8020.337,E2 -8020.337} C_VEL
LIN {X 0,Y 460.842,Z 969.368,A -85,B 0,C 180,E1 -8021.44,E2 -8021.44} C_VEL
LIN {X 0,Y 461.335,Z 959.622,A -85,B 0,C 180,E1 -8022.457,E2 -8022.457} C_VEL
LIN {X 0,Y 461.838,Z 948.161,A -85,B 0,C 180,E1 -8023.424,E2 -8023.424} C_VEL
LIN {X 0,Y 462.316,Z 936.641,A -85,B 0,C 180,E1 -8024.194,E2 -8024.194} C_VEL
LIN {X 0,Y 462.834,Z 924.841,A -85,B 0,C 180,E1 -8024.796,E2 -8024.796} C_VEL
LIN {X 0,Y 463.312,Z 911.267,A -85,B 0,C 180,E1 -8025.286,E2 -8025.286} C_VEL
LIN {X 0,Y 463.621,Z 897.784,A -85,B 0,C 180,E1 -8025.586,E2 -8025.586} C_VEL
LIN {X 0,Y 464.245,Z 817.24,A -85,B 0,C 180,E1 -8026.83,E2 -8026.83} C_VEL
LIN {X 0,Y 461.564,Z 793.449,A -85,B 0,C 180,E1 -8027.306,E2 -8027.306} C_VEL
LIN {X 0,Y 462.426,Z 771.484,A -85,B 0,C 180,E1 -8030.233,E2 -8030.233} C_VEL
LIN {X 0,Y 463.405,Z 747.185,A -85,B 0,C 180,E1 -8033.464,E2 -8033.464} C_VEL
LIN {X 0,Y 464.382,Z 724.998,A -85,B 0,C 180,E1 -8036.443,E2 -8036.443} C_VEL
LIN {X 0,Y 464.876,Z 715.674,A -85,B 0,C 180,E1 -8037.707,E2 -8037.707} C_VEL
LIN {X 0,Y 463.909,Z 710.182,A -85,B 0,C 180,E1 -8038.517,E2 -8038.517} C_VEL
LIN {X 0,Y 460.526,Z 695.122,A -85,B 0,C 180,E1 -8040.878,E2 -8040.878} C_VEL
LIN {X 0,Y 460.483,Z 695.126,A -85,B 0,C 180,E1 -8043.333,E2 -8043.333} C_VEL
LIN {X 0,Y 460.446,Z 695.122,A -85,B 0,C 180,E1 -8046.536,E2 -8046.536} C_VEL
LIN {X 0,Y 460.493,Z 695.124,A -85,B 0,C 180,E1 -8048.889,E2 -8048.889} C_VEL
LIN {X 0,Y 460.51,Z 695.121,A -85,B 0,C 180,E1 -8051.599,E2 -8051.599} C_VEL
LIN {X 0,Y 460.513,Z 695.119,A -85,B 0,C 180,E1 -8054.593,E2 -8054.593} C_VEL
LIN {X 0,Y 460.489,Z 695.122,A -85,B 0,C 180,E1 -8057.815,E2 -8057.815} C_VEL
LIN {X 0,Y 460.525,Z 695.117,A -85,B 0,C 180,E1 -8060.137,E2 -8060.137} C_VEL
LIN {X 0,Y 460.48,Z 695.128,A -85,B 0,C 180,E1 -8063.471,E2 -8063.471} C_VEL
LIN {X 0,Y 460.535,Z 695.116,A -85,B 0,C 180,E1 -8066.675,E2 -8066.675} C_VEL
LIN {X 0,Y 460.521,Z 695.12,A -85,B 0,C 180,E1 -8069.761,E2 -8069.761} C_VEL
LIN {X 0,Y 460.53,Z 695.119,A -85,B 0,C 180,E1 -8072.753,E2 -8072.753} C_VEL
LIN {X 0,Y 460.537,Z 695.12,A -85,B 0,C 180,E1 -8075.667,E2 -8075.667} C_VEL
LIN {X 0,Y 460.537,Z 695.118,A -85,B 0,C 180,E1 -8078.579,E2 -8078.579} C_VEL
LIN {X 0,Y 460.6,Z 695.115,A -85,B 0,C 180,E1 -8081.311,E2 -8081.311} C_VEL
LIN {X 0,Y 460.564,Z 695.118,A -85,B 0,C 180,E1 -8083.24,E2 -8083.24} C_VEL
LIN {X 0,Y 464.336,Z 705.485,A -85,B 0,C 180,E1 -8083.617,E2 -8083.617} C_VEL
LIN {X 0,Y 463.607,Z 776.014,A -85,B 0,C 180,E1 -8084.897,E2 -8084.897} C_VEL
LIN {X 0,Y 463.476,Z 788.283,A -85,B 0,C 180,E1 -8085.258,E2 -8085.258} C_VEL
LIN {X 0,Y 463.414,Z 798.293,A -85,B 0,C 180,E1 -8085.677,E2 -8085.677} C_VEL
LIN {X 0,Y 463.136,Z 808.411,A -85,B 0,C 180,E1 -8086.221,E2 -8086.221} C_VEL
LIN {X 0,Y 462.872,Z 817.57,A -85,B 0,C 180,E1 -8086.835,E2 -8086.835} C_VEL
LIN {X 0,Y 462.518,Z 826.94,A -85,B 0,C 180,E1 -8087.606,E2 -8087.606} C_VEL
LIN {X 0,Y 462.243,Z 834.769,A -85,B 0,C 180,E1 -8088.378,E2 -8088.378} C_VEL
LIN {X 0,Y 461.945,Z 842.309,A -85,B 0,C 180,E1 -8089.259,E2 -8089.259} C_VEL
LIN {X 0,Y 461.557,Z 850.116,A -85,B 0,C 180,E1 -8090.358,E2 -8090.358} C_VEL
LIN {X 0,Y 461.281,Z 856.575,A -85,B 0,C 180,E1 -8091.457,E2 -8091.457} C_VEL
LIN {X 0,Y 461.06,Z 862.105,A -85,B 0,C 180,E1 -8092.598,E2 -8092.598} C_VEL
LIN {X 0,Y 460.819,Z 867.064,A -85,B 0,C 180,E1 -8093.872,E2 -8093.872} C_VEL
LIN {X 0,Y 460.578,Z 869.928,A -85,B 0,C 180,E1 -8094.747,E2 -8094.747} C_VEL
LIN {X 0,Y 460.428,Z 873.912,A -85,B 0,C 180,E1 -8096.5,E2 -8096.5} C_VEL
LIN {X 0,Y 460.429,Z 875.359,A -85,B 0,C 180,E1 -8097.375,E2 -8097.375} C_VEL
LIN {X 0,Y 460.339,Z 876.824,A -85,B 0,C 180,E1 -8099.125,E2 -8099.125} C_VEL
LIN {X 0,Y 460.308,Z 876.967,A -85,B 0,C 180,E1 -8100,E2 -8100} C_VEL
LIN {X 0,Y 460.302,Z 876.671,A -85,B 0,C 180,E1 -8100.875,E2 -8100.875} C_VEL
LIN {X 0,Y 460.199,Z 874.895,A -85,B 0,C 180,E1 -8102.626,E2 -8102.626} C_VEL
LIN {X 0,Y 460.383,Z 871.344,A -85,B 0,C 180,E1 -8104.378,E2 -8104.378} C_VEL
LIN {X 0,Y 460.536,Z 867.522,A -85,B 0,C 180,E1 -8105.693,E2 -8105.693} C_VEL
LIN {X 0,Y 460.771,Z 863.664,A -85,B 0,C 180,E1 -8106.746,E2 -8106.746} C_VEL
LIN {X 0,Y 460.965,Z 857.441,A -85,B 0,C 180,E1 -8108.107,E2 -8108.107} C_VEL
LIN {X 0,Y 461.26,Z 851.276,A -85,B 0,C 180,E1 -8109.206,E2 -8109.206} C_VEL
LIN {X 0,Y 461.52,Z 843.842,A -85,B 0,C 180,E1 -8110.307,E2 -8110.307} C_VEL
LIN {X 0,Y 461.843,Z 835.805,A -85,B 0,C 180,E1 -8111.299,E2 -8111.299} C_VEL
LIN {X 0,Y 462.18,Z 827.264,A -85,B 0,C 180,E1 -8112.18,E2 -8112.18} C_VEL
LIN {X 0,Y 462.485,Z 818.309,A -85,B 0,C 180,E1 -8112.953,E2 -8112.953} C_VEL
LIN {X 0,Y 462.749,Z 809.562,A -85,B 0,C 180,E1 -8113.582,E2 -8113.582} C_VEL
LIN {X 0,Y 463.023,Z 798.425,A -85,B 0,C 180,E1 -8114.223,E2 -8114.223} C_VEL
LIN {X 0,Y 463.226,Z 788.585,A -85,B 0,C 180,E1 -8114.666,E2 -8114.666} C_VEL
LIN {X 0,Y 463.326,Z 777.777,A -85,B 0,C 180,E1 -8115.028,E2 -8115.028} C_VEL
LIN {X 0,Y 463.443,Z 765.288,A -85,B 0,C 180,E1 -8115.305,E2 -8115.305} C_VEL
LIN {X 0,Y 463.908,Z 705.233,A -85,B 0,C 180,E1 -8116.329,E2 -8116.329} C_VEL
LIN {X 0,Y 460.569,Z 695.118,A -85,B 0,C 180,E1 -8116.644,E2 -8116.644} C_VEL
LIN {X 0,Y 460.581,Z 695.11,A -85,B 0,C 180,E1 -8119.615,E2 -8119.615} C_VEL
LIN {X 0,Y 460.522,Z 695.119,A -85,B 0,C 180,E1 -8122.428,E2 -8122.428} C_VEL
LIN {X 0,Y 460.561,Z 695.111,A -85,B 0,C 180,E1 -8125.795,E2 -8125.795} C_VEL
LIN {X 0,Y 460.542,Z 695.113,A -85,B 0,C 180,E1 -8128.234,E2 -8128.234} C_VEL
LIN {X 0,Y 460.537,Z 695.117,A -85,B 0,C 180,E1 -8131.282,E2 -8131.282} C_VEL
LIN {X 0,Y 460.538,Z 695.116,A -85,B 0,C 180,E1 -8134.502,E2 -8134.502} C_VEL
LIN {X 0,Y 460.514,Z 695.117,A -85,B 0,C 180,E1 -8137.622,E2 -8137.622} C_VEL
LIN {X 0,Y 460.533,Z 695.12,A -85,B 0,C 180,E1 -8141.011,E2 -8141.011} C_VEL
LIN {X 0,Y 460.527,Z 695.115,A -85,B 0,C 180,E1 -8144.588,E2 -8144.588} C_VEL
LIN {X 0,Y 460.49,Z 695.118,A -85,B 0,C 180,E1 -8147.811,E2 -8147.811} C_VEL
LIN {X 0,Y 460.525,Z 695.113,A -85,B 0,C 180,E1 -8150.133,E2 -8150.133} C_VEL
LIN {X 0,Y 460.473,Z 695.124,A -85,B 0,C 180,E1 -8153.466,E2 -8153.466} C_VEL
LIN {X 0,Y 460.516,Z 695.117,A -85,B 0,C 180,E1 -8156.67,E2 -8156.67} C_VEL
LIN {X 0,Y 460.493,Z 695.12,A -85,B 0,C 180,E1 -8159.754,E2 -8159.754} C_VEL
LIN {X 0,Y 460.494,Z 695.12,A -85,B 0,C 180,E1 -8162.747,E2 -8162.747} C_VEL
LIN {X 0,Y 460.507,Z 695.122,A -85,B 0,C 180,E1 -8165.661,E2 -8165.661} C_VEL
LIN {X 0,Y 460.507,Z 695.12,A -85,B 0,C 180,E1 -8168.32,E2 -8168.32} C_VEL
LIN {X 0,Y 459.868,Z 695.204,A -85,B 0,C 180,E1 -8169.051,E2 -8169.051} C_VEL
LIN {X 0,Y 457.005,Z 695.559,A -85,B 0,C 180,E1 -8170.236,E2 -8170.236} C_VEL
LIN {X 0,Y 454.579,Z 695.864,A -85,B 0,C 180,E1 -8171.193,E2 -8171.193} C_VEL
LIN {X 0,Y 453.555,Z 695.989,A -85,B 0,C 180,E1 -8171.932,E2 -8171.932} C_VEL
LIN {X 0,Y 453.483,Z 695.997,A -85,B 0,C 180,E1 -8172.182,E2 -8172.182} C_VEL
LIN {X 0,Y 453.489,Z 696.03,A -85,B 0,C 180,E1 -8172.87,E2 -8172.87} C_VEL
LIN {X 0,Y 457.879,Z 708.099,A -85,B 0,C 180,E1 -8173.245,E2 -8173.245} C_VEL
LIN {X 0,Y 457.394,Z 777.636,A -85,B 0,C 180,E1 -8174.368,E2 -8174.368} C_VEL
LIN {X 0,Y 457.407,Z 790.732,A -85,B 0,C 180,E1 -8174.768,E2 -8174.768} C_VEL
LIN {X 0,Y 457.165,Z 802.752,A -85,B 0,C 180,E1 -8175.302,E2 -8175.302} C_VEL
LIN {X 0,Y 456.836,Z 814.308,A -85,B 0,C 180,E1 -8175.991,E2 -8175.991} C_VEL
LIN {X 0,Y 456.338,Z 825.61,A -85,B 0,C 180,E1 -8176.865,E2 -8176.865} C_VEL
LIN {X 0,Y 455.874,Z 835.955,A -85,B 0,C 180,E1 -8177.87,E2 -8177.87} C_VEL
LIN {X 0,Y 455.481,Z 844.386,A -85,B 0,C 180,E1 -8178.874,E2 -8178.874} C_VEL
LIN {X 0,Y 454.991,Z 852.154,A -85,B 0,C 180,E1 -8179.988,E2 -8179.988} C_VEL
LIN {X 0,Y 454.518,Z 859.845,A -85,B 0,C 180,E1 -8181.346,E2 -8181.346} C_VEL
LIN {X 0,Y 454.267,Z 865.496,A -85,B 0,C 180,E1 -8182.59,E2 -8182.59} C_VEL
LIN {X 0,Y 453.941,Z 871.27,A -85,B 0,C 180,E1 -8184.219,E2 -8184.219} C_VEL
LIN {X 0,Y 453.59,Z 874.819,A -85,B 0,C 180,E1 -8185.551,E2 -8185.551} C_VEL
LIN {X 0,Y 453.468,Z 876.644,A -85,B 0,C 180,E1 -8186.44,E2 -8186.44} C_VEL
LIN {X 0,Y 453.465,Z 878.011,A -85,B 0,C 180,E1 -8187.329,E2 -8187.329} C_VEL
LIN {X 0,Y 453.409,Z 879.588,A -85,B 0,C 180,E1 -8189.106,E2 -8189.106} C_VEL
LIN {X 0,Y 453.386,Z 879.824,A -85,B 0,C 180,E1 -8189.994,E2 -8189.994} C_VEL
LIN {X 0,Y 453.503,Z 879.068,A -85,B 0,C 180,E1 -8191.77,E2 -8191.77} C_VEL
LIN {X 0,Y 453.458,Z 876.834,A -85,B 0,C 180,E1 -8193.548,E2 -8193.548} C_VEL
LIN {X 0,Y 453.668,Z 874.028,A -85,B 0,C 180,E1 -8194.881,E2 -8194.881} C_VEL
LIN {X 0,Y 453.978,Z 870.217,A -85,B 0,C 180,E1 -8196.215,E2 -8196.215} C_VEL
LIN {X 0,Y 454.24,Z 864.745,A -85,B 0,C 180,E1 -8197.689,E2 -8197.689} C_VEL
LIN {X 0,Y 454.639,Z 857.941,A -85,B 0,C 180,E1 -8199.11,E2 -8199.11} C_VEL
LIN {X 0,Y 455.152,Z 849.928,A -85,B 0,C 180,E1 -8200.446,E2 -8200.446} C_VEL
LIN {X 0,Y 455.628,Z 841.715,A -85,B 0,C 180,E1 -8201.561,E2 -8201.561} C_VEL
LIN {X 0,Y 456.077,Z 831.565,A -85,B 0,C 180,E1 -8202.678,E2 -8202.678} C_VEL
LIN {X 0,Y 456.632,Z 821.115,A -85,B 0,C 180,E1 -8203.597,E2 -8203.597} C_VEL
LIN {X 0,Y 457.024,Z 809.35,A -85,B 0,C 180,E1 -8204.421,E2 -8204.421} C_VEL
LIN {X 0,Y 457.264,Z 796.859,A -85,B 0,C 180,E1 -8205.076,E2 -8205.076} C_VEL
LIN {X 0,Y 457.441,Z 783.764,A -85,B 0,C 180,E1 -8205.561,E2 -8205.561} C_VEL
LIN {X 0,Y 457.439,Z 771.394,A -85,B 0,C 180,E1 -8205.847,E2 -8205.847} C_VEL
LIN {X 0,Y 457.906,Z 708.146,A -85,B 0,C 180,E1 -8206.847,E2 -8206.847} C_VEL
LIN {X 0,Y 453.511,Z 695.999,A -85,B 0,C 180,E1 -8207.233,E2 -8207.233} C_VEL
LIN {X 0,Y 453.487,Z 695.995,A -85,B 0,C 180,E1 -8209.927,E2 -8209.927} C_VEL
LIN {X 0,Y 453.458,Z 695.996,A -85,B 0,C 180,E1 -8212.789,E2 -8212.789} C_VEL
LIN {X 0,Y 453.473,Z 695.991,A -85,B 0,C 180,E1 -8215.986,E2 -8215.986} C_VEL
LIN {X 0,Y 453.48,Z 695.994,A -85,B 0,C 180,E1 -8218.705,E2 -8218.705} C_VEL
LIN {X 0,Y 453.433,Z 696.002,A -85,B 0,C 180,E1 -8221.793,E2 -8221.793} C_VEL
LIN {X 0,Y 453.446,Z 696,A -85,B 0,C 180,E1 -8224.982,E2 -8224.982} C_VEL
LIN {X 0,Y 453.441,Z 695.988,A -85,B 0,C 180,E1 -8228.303,E2 -8228.303} C_VEL
LIN {X 0,Y 453.475,Z 695.995,A -85,B 0,C 180,E1 -8230.6,E2 -8230.6} C_VEL
LIN {X 0,Y 453.437,Z 696.004,A -85,B 0,C 180,E1 -8233.241,E2 -8233.241} C_VEL
LIN {X 0,Y 453.428,Z 695.996,A -85,B 0,C 180,E1 -8235.774,E2 -8235.774} C_VEL
LIN {X 0,Y 453.446,Z 696.002,A -85,B 0,C 180,E1 -8238.205,E2 -8238.205} C_VEL
LIN {X 0,Y 453.483,Z 695.991,A -85,B 0,C 180,E1 -8240.781,E2 -8240.781} C_VEL
LIN {X 0,Y 453.4,Z 696.011,A -85,B 0,C 180,E1 -8243.912,E2 -8243.912} C_VEL
LIN {X 0,Y 453.423,Z 695.999,A -85,B 0,C 180,E1 -8247.146,E2 -8247.146} C_VEL
LIN {X 0,Y 453.451,Z 695.997,A -85,B 0,C 180,E1 -8250.266,E2 -8250.266} C_VEL
LIN {X 0,Y 453.449,Z 695.996,A -85,B 0,C 180,E1 -8253.29,E2 -8253.29} C_VEL
LIN {X 0,Y 453.437,Z 696,A -85,B 0,C 180,E1 -8256.235,E2 -8256.235} C_VEL
LIN {X 0,Y 453.413,Z 696.002,A -85,B 0,C 180,E1 -8259.114,E2 -8259.114} C_VEL
LIN {X 0,Y 453.44,Z 695.997,A -85,B 0,C 180,E1 -8261.941,E2 -8261.941} C_VEL
LIN {X 0,Y 453.482,Z 695.999,A -85,B 0,C 180,E1 -8264.724,E2 -8264.724} C_VEL
LIN {X 0,Y 453.528,Z 695.986,A -85,B 0,C 180,E1 -8267.47,E2 -8267.47} C_VEL
LIN {X 0,Y 453.523,Z 695.992,A -85,B 0,C 180,E1 -8271.085,E2 -8271.085} C_VEL
LIN {X 0,Y 453.608,Z 695.978,A -85,B 0,C 180,E1 -8273.774,E2 -8273.774} C_VEL
LIN {X 0,Y 453.699,Z 695.969,A -85,B 0,C 180,E1 -8277.336,E2 -8277.336} C_VEL
LIN {X 0,Y 453.745,Z 695.962,A -85,B 0,C 180,E1 -8280,E2 -8280} C_VEL
LIN {X 0,Y 453.7,Z 695.966,A -85,B 0,C 180,E1 -8282.664,E2 -8282.664} C_VEL
LIN {X 0,Y 453.608,Z 695.979,A -85,B 0,C 180,E1 -8286.226,E2 -8286.226} C_VEL
LIN {X 0,Y 453.523,Z 695.989,A -85,B 0,C 180,E1 -8288.915,E2 -8288.915} C_VEL
LIN {X 0,Y 453.527,Z 695.988,A -85,B 0,C 180,E1 -8292.553,E2 -8292.553} C_VEL
LIN {X 0,Y 453.483,Z 695.992,A -85,B 0,C 180,E1 -8296.198,E2 -8296.198} C_VEL
LIN {X 0,Y 453.448,Z 695.999,A -85,B 0,C 180,E1 -8299.044,E2 -8299.044} C_VEL
LIN {X 0,Y 453.409,Z 696.007,A -85,B 0,C 180,E1 -8301.84,E2 -8301.84} C_VEL
LIN {X 0,Y 453.462,Z 695.994,A -85,B 0,C 180,E1 -8304.737,E2 -8304.737} C_VEL
LIN {X 0,Y 453.473,Z 696,A -85,B 0,C 180,E1 -8307.966,E2 -8307.966} C_VEL
LIN {X 0,Y 453.421,Z 695.998,A -85,B 0,C 180,E1 -8310.764,E2 -8310.764} C_VEL
LIN {X 0,Y 453.418,Z 696.005,A -85,B 0,C 180,E1 -8313.918,E2 -8313.918} C_VEL
LIN {X 0,Y 453.416,Z 696,A -85,B 0,C 180,E1 -8317.193,E2 -8317.193} C_VEL
LIN {X 0,Y 453.484,Z 695.985,A -85,B 0,C 180,E1 -8319.45,E2 -8319.45} C_VEL
LIN {X 0,Y 453.442,Z 695.999,A -85,B 0,C 180,E1 -8322.998,E2 -8322.998} C_VEL
LIN {X 0,Y 453.43,Z 696.002,A -85,B 0,C 180,E1 -8325.787,E2 -8325.787} C_VEL
LIN {X 0,Y 453.453,Z 695.997,A -85,B 0,C 180,E1 -8328.218,E2 -8328.218} C_VEL
LIN {X 0,Y 453.489,Z 695.995,A -85,B 0,C 180,E1 -8330.794,E2 -8330.794} C_VEL
LIN {X 0,Y 453.419,Z 696.002,A -85,B 0,C 180,E1 -8333.924,E2 -8333.924} C_VEL
LIN {X 0,Y 453.45,Z 695.996,A -85,B 0,C 180,E1 -8337.158,E2 -8337.158} C_VEL
LIN {X 0,Y 453.494,Z 696.168,A -85,B 0,C 180,E1 -8338.914,E2 -8338.914} C_VEL
LIN {X 0,Y 457.357,Z 713.021,A -85,B 0,C 180,E1 -8341.561,E2 -8341.561} C_VEL
LIN {X 0,Y 457.955,Z 716.623,A -85,B 0,C 180,E1 -8342.1,E2 -8342.1} C_VEL
LIN {X 0,Y 456.947,Z 737.053,A -85,B 0,C 180,E1 -8344.907,E2 -8344.907} C_VEL
LIN {X 0,Y 455.907,Z 760.669,A -85,B 0,C 180,E1 -8348.112,E2 -8348.112} C_VEL
LIN {X 0,Y 454.798,Z 787.68,A -85,B 0,C 180,E1 -8351.772,E2 -8351.772} C_VEL
LIN {X 0,Y 454.584,Z 792.433,A -85,B 0,C 180,E1 -8352.418,E2 -8352.418} C_VEL
LIN {X 0,Y 457.421,Z 818.994,A -85,B 0,C 180,E1 -8352.955,E2 -8352.955} C_VEL
LIN {X 0,Y 456.689,Z 903.268,A -85,B 0,C 180,E1 -8354.298,E2 -8354.298} C_VEL
LIN {X 0,Y 456.258,Z 916.511,A -85,B 0,C 180,E1 -8354.684,E2 -8354.684} C_VEL
LIN {X 0,Y 455.758,Z 928.72,A -85,B 0,C 180,E1 -8355.21,E2 -8355.21} C_VEL
LIN {X 0,Y 455.086,Z 941.08,A -85,B 0,C 180,E1 -8355.93,E2 -8355.93} C_VEL
LIN {X 0,Y 454.593,Z 952.385,A -85,B 0,C 180,E1 -8356.788,E2 -8356.788} C_VEL
LIN {X 0,Y 454.116,Z 963.418,A -85,B 0,C 180,E1 -8357.834,E2 -8357.834} C_VEL
LIN {X 0,Y 453.651,Z 972.099,A -85,B 0,C 180,E1 -8358.841,E2 -8358.841} C_VEL
LIN {X 0,Y 453.272,Z 980.132,A -85,B 0,C 180,E1 -8359.961,E2 -8359.961} C_VEL
LIN {X 0,Y 453.034,Z 988.015,A -85,B 0,C 180,E1 -8361.307,E2 -8361.307} C_VEL
LIN {X 0,Y 452.853,Z 995.294,A -85,B 0,C 180,E1 -8362.874,E2 -8362.874} C_VEL
LIN {X 0,Y 452.81,Z 1000.155,A -85,B 0,C 180,E1 -8364.216,E2 -8364.216} C_VEL
LIN {X 0,Y 452.787,Z 1003.878,A -85,B 0,C 180,E1 -8365.555,E2 -8365.555} C_VEL
LIN {X 0,Y 452.812,Z 1005.802,A -85,B 0,C 180,E1 -8366.447,E2 -8366.447} C_VEL
LIN {X 0,Y 452.778,Z 1007.236,A -85,B 0,C 180,E1 -8367.337,E2 -8367.337} C_VEL
LIN {X 0,Y 452.775,Z 1008.262,A -85,B 0,C 180,E1 -8368.227,E2 -8368.227} C_VEL
LIN {X 0,Y 452.761,Z 1008.885,A -85,B 0,C 180,E1 -8369.117,E2 -8369.117} C_VEL
LIN {X 0,Y 452.763,Z 1009.104,A -85,B 0,C 180,E1 -8370.006,E2 -8370.006} C_VEL
LIN {X 0,Y 452.761,Z 1008.878,A -85,B 0,C 180,E1 -8370.895,E2 -8370.895} C_VEL
LIN {X 0,Y 452.776,Z 1008.249,A -85,B 0,C 180,E1 -8371.785,E2 -8371.785} C_VEL
LIN {X 0,Y 452.78,Z 1007.219,A -85,B 0,C 180,E1 -8372.675,E2 -8372.675} C_VEL
LIN {X 0,Y 452.816,Z 1005.777,A -85,B 0,C 180,E1 -8373.565,E2 -8373.565} C_VEL
LIN {X 0,Y 452.805,Z 1002.744,A -85,B 0,C 180,E1 -8374.903,E2 -8374.903} C_VEL
LIN {X 0,Y 452.817,Z 998.643,A -85,B 0,C 180,E1 -8376.243,E2 -8376.243} C_VEL
LIN {X 0,Y 452.911,Z 992.345,A -85,B 0,C 180,E1 -8377.809,E2 -8377.809} C_VEL
LIN {X 0,Y 453.105,Z 985.491,A -85,B 0,C 180,E1 -8379.153,E2 -8379.153} C_VEL
LIN {X 0,Y 453.398,Z 977.011,A -85,B 0,C 180,E1 -8380.499,E2 -8380.499} C_VEL
LIN {X 0,Y 453.795,Z 968.341,A -85,B 0,C 180,E1 -8381.62,E2 -8381.62} C_VEL
LIN {X 0,Y 454.295,Z 958.429,A -85,B 0,C 180,E1 -8382.668,E2 -8382.668} C_VEL
LIN {X 0,Y 454.877,Z 947.138,A -85,B 0,C 180,E1 -8383.633,E2 -8383.633} C_VEL
LIN {X 0,Y 455.403,Z 935.621,A -85,B 0,C 180,E1 -8384.414,E2 -8384.414} C_VEL
LIN {X 0,Y 455.939,Z 923.819,A -85,B 0,C 180,E1 -8385.025,E2 -8385.025} C_VEL
LIN {X 0,Y 456.499,Z 910.254,A -85,B 0,C 180,E1 -8385.52,E2 -8385.52} C_VEL
LIN {X 0,Y 456.768,Z 896.756,A -85,B 0,C 180,E1 -8385.826,E2 -8385.826} C_VEL
LIN {X 0,Y 457.417,Z 817.88,A -85,B 0,C 180,E1 -8387.062,E2 -8387.062} C_VEL
LIN {X 0,Y 454.616,Z 792.285,A -85,B 0,C 180,E1 -8387.6,E2 -8387.6} C_VEL
LIN {X 0,Y 455.602,Z 767.065,A -85,B 0,C 180,E1 -8391.022,E2 -8391.022} C_VEL
LIN {X 0,Y 456.61,Z 744.49,A -85,B 0,C 180,E1 -8394.076,E2 -8394.076} C_VEL
LIN {X 0,Y 457.82,Z 720.02,A -85,B 0,C 180,E1 -8397.426,E2 -8397.426} C_VEL
LIN {X 0,Y 457.955,Z 716.516,A -85,B 0,C 180,E1 -8397.913,E2 -8397.913} C_VEL
LIN {X 0,Y 454.613,Z 700.973,A -85,B 0,C 180,E1 -8400.314,E2 -8400.314} C_VEL
LIN {X 0,Y 453.484,Z 696.001,A -85,B 0,C 180,E1 -8401.127,E2 -8401.127} C_VEL
LIN {X 0,Y 453.422,Z 696.006,A -85,B 0,C 180,E1 -8403.922,E2 -8403.922} C_VEL
LIN {X 0,Y 453.437,Z 696.003,A -85,B 0,C 180,E1 -8407.196,E2 -8407.196} C_VEL
LIN {X 0,Y 453.48,Z 695.996,A -85,B 0,C 180,E1 -8410.615,E2 -8410.615} C_VEL
LIN {X 0,Y 453.456,Z 695.997,A -85,B 0,C 180,E1 -8414.227,E2 -8414.227} C_VEL
LIN {X 0,Y 453.431,Z 696.003,A -85,B 0,C 180,E1 -8417.001,E2 -8417.001} C_VEL
LIN {X 0,Y 453.487,Z 695.999,A -85,B 0,C 180,E1 -8419.415,E2 -8419.415} C_VEL
LIN {X 0,Y 453.454,Z 696,A -85,B 0,C 180,E1 -8422.81,E2 -8422.81} C_VEL
LIN {X 0,Y 453.483,Z 695.994,A -85,B 0,C 180,E1 -8426.088,E2 -8426.088} C_VEL
LIN {X 0,Y 453.482,Z 696.001,A -85,B 0,C 180,E1 -8429.241,E2 -8429.241} C_VEL
LIN {X 0,Y 453.506,Z 695.993,A -85,B 0,C 180,E1 -8432.295,E2 -8432.295} C_VEL
LIN {X 0,Y 453.509,Z 695.997,A -85,B 0,C 180,E1 -8435.265,E2 -8435.265} C_VEL
LIN {X 0,Y 453.496,Z 695.995,A -85,B 0,C 180,E1 -8438.416,E2 -8438.416} C_VEL
LIN {X 0,Y 453.539,Z 695.993,A -85,B 0,C 180,E1 -8441.009,E2 -8441.009} C_VEL
LIN {X 0,Y 453.517,Z 695.995,A -85,B 0,C 180,E1 -8442.928,E2 -8442.928} C_VEL
LIN {X 0,Y 457.726,Z 707.446,A -85,B 0,C 180,E1 -8443.356,E2 -8443.356} C_VEL
LIN {X 0,Y 456.845,Z 777.198,A -85,B 0,C 180,E1 -8444.668,E2 -8444.668} C_VEL
LIN {X 0,Y 456.704,Z 789.44,A -85,B 0,C 180,E1 -8445.034,E2 -8445.034} C_VEL
LIN {X 0,Y 456.605,Z 799.463,A -85,B 0,C 180,E1 -8445.459,E2 -8445.459} C_VEL
LIN {X 0,Y 456.362,Z 809.192,A -85,B 0,C 180,E1 -8445.986,E2 -8445.986} C_VEL
LIN {X 0,Y 456.058,Z 818.751,A -85,B 0,C 180,E1 -8446.635,E2 -8446.635} C_VEL
LIN {X 0,Y 455.688,Z 828.128,A -85,B 0,C 180,E1 -8447.417,E2 -8447.417} C_VEL
LIN {X 0,Y 455.409,Z 835.96,A -85,B 0,C 180,E1 -8448.201,E2 -8448.201} C_VEL
LIN {X 0,Y 455.075,Z 843.506,A -85,B 0,C 180,E1 -8449.095,E2 -8449.095} C_VEL
LIN {X 0,Y 454.671,Z 851.295,A -85,B 0,C 180,E1 -8450.21,E2 -8450.21} C_VEL
LIN {X 0,Y 454.375,Z 857.731,A -85,B 0,C 180,E1 -8451.326,E2 -8451.326} C_VEL
LIN {X 0,Y 454.128,Z 863.102,A -85,B 0,C 180,E1 -8452.45,E2 -8452.45} C_VEL
LIN {X 0,Y 453.849,Z 868.184,A -85,B 0,C 180,E1 -8453.777,E2 -8453.777} C_VEL
LIN {X 0,Y 453.596,Z 871.042,A -85,B 0,C 180,E1 -8454.666,E2 -8454.666} C_VEL
LIN {X 0,Y 453.449,Z 875.011,A -85,B 0,C 180,E1 -8456.446,E2 -8456.446} C_VEL
LIN {X 0,Y 453.443,Z 876.45,A -85,B 0,C 180,E1 -8457.335,E2 -8457.335} C_VEL
LIN {X 0,Y 453.327,Z 877.891,A -85,B 0,C 180,E1 -8459.112,E2 -8459.112} C_VEL
LIN {X 0,Y 453.296,Z 878.02,A -85,B 0,C 180,E1 -8460,E2 -8460} C_VEL
LIN {X 0,Y 453.292,Z 877.702,A -85,B 0,C 180,E1 -8460.888,E2 -8460.888} C_VEL
LIN {X 0,Y 453.177,Z 875.887,A -85,B 0,C 180,E1 -8462.667,E2 -8462.667} C_VEL
LIN {X 0,Y 453.366,Z 872.273,A -85,B 0,C 180,E1 -8464.445,E2 -8464.445} C_VEL
LIN {X 0,Y 453.54,Z 868.4,A -85,B 0,C 180,E1 -8465.781,E2 -8465.781} C_VEL
LIN {X 0,Y 453.763,Z 864.835,A -85,B 0,C 180,E1 -8466.771,E2 -8466.771} C_VEL
LIN {X 0,Y 453.99,Z 858.203,A -85,B 0,C 180,E1 -8468.233,E2 -8468.233} C_VEL
LIN {X 0,Y 454.303,Z 851.969,A -85,B 0,C 180,E1 -8469.348,E2 -8469.348} C_VEL
LIN {X 0,Y 454.577,Z 844.457,A -85,B 0,C 180,E1 -8470.467,E2 -8470.467} C_VEL
LIN {X 0,Y 454.914,Z 836.33,A -85,B 0,C 180,E1 -8471.473,E2 -8471.473} C_VEL
LIN {X 0,Y 455.215,Z 828.881,A -85,B 0,C 180,E1 -8472.256,E2 -8472.256} C_VEL
LIN {X 0,Y 455.528,Z 820.047,A -85,B 0,C 180,E1 -8473.041,E2 -8473.041} C_VEL
LIN {X 0,Y 455.834,Z 810.426,A -85,B 0,C 180,E1 -8473.745,E2 -8473.745} C_VEL
LIN {X 0,Y 456.074,Z 800.579,A -85,B 0,C 180,E1 -8474.331,E2 -8474.331} C_VEL
LIN {X 0,Y 456.316,Z 789.642,A -85,B 0,C 180,E1 -8474.836,E2 -8474.836} C_VEL
LIN {X 0,Y 456.434,Z 778.911,A -85,B 0,C 180,E1 -8475.203,E2 -8475.203} C_VEL
LIN {X 0,Y 456.531,Z 766.591,A -85,B 0,C 180,E1 -8475.486,E2 -8475.486} C_VEL
LIN {X 0,Y 457.061,Z 706.612,A -85,B 0,C 180,E1 -8476.532,E2 -8476.532} C_VEL
LIN {X 0,Y 453.542,Z 695.993,A -85,B 0,C 180,E1 -8476.858,E2 -8476.858} C_VEL
LIN {X 0,Y 453.517,Z 695.99,A -85,B 0,C 180,E1 -8479.933,E2 -8479.933} C_VEL
LIN {X 0,Y 453.491,Z 695.999,A -85,B 0,C 180,E1 -8482.795,E2 -8482.795} C_VEL
LIN {X 0,Y 453.509,Z 695.99,A -85,B 0,C 180,E1 -8485.991,E2 -8485.991} C_VEL
LIN {X 0,Y 453.508,Z 695.995,A -85,B 0,C 180,E1 -8488.712,E2 -8488.712} C_VEL
LIN {X 0,Y 453.477,Z 695.994,A -85,B 0,C 180,E1 -8491.799,E2 -8491.799} C_VEL
LIN {X 0,Y 453.491,Z 695.998,A -85,B 0,C 180,E1 -8494.989,E2 -8494.989} C_VEL
LIN {X 0,Y 453.473,Z 695.994,A -85,B 0,C 180,E1 -8498.311,E2 -8498.311} C_VEL
LIN {X 0,Y 453.487,Z 695.994,A -85,B 0,C 180,E1 -8500.61,E2 -8500.61} C_VEL
LIN {X 0,Y 453.475,Z 695.991,A -85,B 0,C 180,E1 -8504.22,E2 -8504.22} C_VEL
LIN {X 0,Y 453.432,Z 696.003,A -85,B 0,C 180,E1 -8506.997,E2 -8506.997} C_VEL
LIN {X 0,Y 453.488,Z 695.994,A -85,B 0,C 180,E1 -8509.41,E2 -8509.41} C_VEL
LIN {X 0,Y 453.45,Z 695.998,A -85,B 0,C 180,E1 -8512.806,E2 -8512.806} C_VEL
LIN {X 0,Y 453.47,Z 695.992,A -85,B 0,C 180,E1 -8516.082,E2 -8516.082} C_VEL
LIN {X 0,Y 453.462,Z 696,A -85,B 0,C 180,E1 -8519.235,E2 -8519.235} C_VEL
LIN {X 0,Y 453.481,Z 695.991,A -85,B 0,C 180,E1 -8522.289,E2 -8522.289} C_VEL
LIN {X 0,Y 453.462,Z 696.001,A -85,B 0,C 180,E1 -8525.258,E2 -8525.258} C_VEL
LIN {X 0,Y 453.488,Z 695.994,A -85,B 0,C 180,E1 -8528.414,E2 -8528.414} C_VEL
LIN {X 0,Y 453.476,Z 695.999,A -85,B 0,C 180,E1 -8531.938,E2 -8531.938} C_VEL
LIN {X 0,Y 453.483,Z 695.997,A -85,B 0,C 180,E1 -8532.182,E2 -8532.182} C_VEL
LIN {X 0,Y 453.496,Z 696.801,A -85,B 0,C 180,E1 -8532.478,E2 -8532.478} C_VEL
LIN {X 0,Y 453.493,Z 699.176,A -85,B 0,C 180,E1 -8532.76,E2 -8532.76} C_VEL
LIN {X 0,Y 453.433,Z 702.308,A -85,B 0,C 180,E1 -8532.945,E2 -8532.945} C_VEL
LIN {X 0,Y 452.994,Z 710.205,A -85,B 0,C 180,E1 -8533.081,E2 -8533.081} C_VEL
LIN {X 0,Y 451.565,Z 721.632,A -85,B 0,C 180,E1 -8533.21,E2 -8533.21} C_VEL
LIN {X 0,Y 451,Z 726.462,A -85,B 0,C 180,E1 -8533.266,E2 -8533.266} C_VEL
LIN {X 0,Y 450.619,Z 778.658,A -85,B 0,C 180,E1 -8534.127,E2 -8534.127} C_VEL
LIN {X 0,Y 450.63,Z 791.746,A -85,B 0,C 180,E1 -8534.533,E2 -8534.533} C_VEL
LIN {X 0,Y 450.37,Z 803.763,A -85,B 0,C 180,E1 -8535.075,E2 -8535.075} C_VEL
LIN {X 0,Y 450.021,Z 815.312,A -85,B 0,C 180,E1 -8535.775,E2 -8535.775} C_VEL
LIN {X 0,Y 449.497,Z 826.618,A -85,B 0,C 180,E1 -8536.661,E2 -8536.661} C_VEL
LIN {X 0,Y 449.007,Z 836.962,A -85,B 0,C 180,E1 -8537.681,E2 -8537.681} C_VEL
LIN {X 0,Y 448.596,Z 845.391,A -85,B 0,C 180,E1 -8538.701,E2 -8538.701} C_VEL
LIN {X 0,Y 448.075,Z 853.159,A -85,B 0,C 180,E1 -8539.831,E2 -8539.831} C_VEL
LIN {X 0,Y 447.575,Z 860.85,A -85,B 0,C 180,E1 -8541.211,E2 -8541.211} C_VEL
LIN {X 0,Y 447.299,Z 866.5,A -85,B 0,C 180,E1 -8542.474,E2 -8542.474} C_VEL
LIN {X 0,Y 446.967,Z 872.272,A -85,B 0,C 180,E1 -8544.128,E2 -8544.128} C_VEL
LIN {X 0,Y 446.583,Z 875.822,A -85,B 0,C 180,E1 -8545.481,E2 -8545.481} C_VEL
LIN {X 0,Y 446.453,Z 877.648,A -85,B 0,C 180,E1 -8546.384,E2 -8546.384} C_VEL
LIN {X 0,Y 446.449,Z 879.014,A -85,B 0,C 180,E1 -8547.287,E2 -8547.287} C_VEL
LIN {X 0,Y 446.389,Z 880.59,A -85,B 0,C 180,E1 -8549.092,E2 -8549.092} C_VEL
LIN {X 0,Y 446.363,Z 880.826,A -85,B 0,C 180,E1 -8549.994,E2 -8549.994} C_VEL
LIN {X 0,Y 446.486,Z 880.07,A -85,B 0,C 180,E1 -8551.798,E2 -8551.798} C_VEL
LIN {X 0,Y 446.443,Z 877.836,A -85,B 0,C 180,E1 -8553.604,E2 -8553.604} C_VEL
LIN {X 0,Y 446.665,Z 875.03,A -85,B 0,C 180,E1 -8554.958,E2 -8554.958} C_VEL
LIN {X 0,Y 446.998,Z 871.217,A -85,B 0,C 180,E1 -8556.312,E2 -8556.312} C_VEL
LIN {X 0,Y 447.276,Z 865.745,A -85,B 0,C 180,E1 -8557.81,E2 -8557.81} C_VEL
LIN {X 0,Y 447.701,Z 858.941,A -85,B 0,C 180,E1 -8559.253,E2 -8559.253} C_VEL
LIN {X 0,Y 448.244,Z 850.927,A -85,B 0,C 180,E1 -8560.609,E2 -8560.609} C_VEL
LIN {X 0,Y 448.746,Z 842.714,A -85,B 0,C 180,E1 -8561.741,E2 -8561.741} C_VEL
LIN {X 0,Y 449.223,Z 832.563,A -85,B 0,C 180,E1 -8562.875,E2 -8562.875} C_VEL
LIN {X 0,Y 449.804,Z 822.112,A -85,B 0,C 180,E1 -8563.807,E2 -8563.807} C_VEL
LIN {X 0,Y 450.199,Z 810.868,A -85,B 0,C 180,E1 -8564.61,E2 -8564.61} C_VEL
LIN {X 0,Y 450.449,Z 799.014,A -85,B 0,C 180,E1 -8565.258,E2 -8565.258} C_VEL
LIN {X 0,Y 450.641,Z 785.663,A -85,B 0,C 180,E1 -8565.773,E2 -8565.773} C_VEL
LIN {X 0,Y 450.65,Z 772.374,A -85,B 0,C 180,E1 -8566.092,E2 -8566.092} C_VEL
LIN {X 0,Y 451.063,Z 709.509,A -85,B 0,C 180,E1 -8567.104,E2 -8567.104} C_VEL
LIN {X 0,Y 446.461,Z 696.875,A -85,B 0,C 180,E1 -8567.514,E2 -8567.514} C_VEL
LIN {X 0,Y 446.427,Z 696.876,A -85,B 0,C 180,E1 -8570.256,E2 -8570.256} C_VEL
LIN {X 0,Y 446.404,Z 696.878,A -85,B 0,C 180,E1 -8573.17,E2 -8573.17} C_VEL
LIN {X 0,Y 446.434,Z 696.868,A -85,B 0,C 180,E1 -8576.191,E2 -8576.191} C_VEL
LIN {X 0,Y 446.419,Z 696.878,A -85,B 0,C 180,E1 -8579.202,E2 -8579.202} C_VEL
LIN {X 0,Y 446.39,Z 696.877,A -85,B 0,C 180,E1 -8582.355,E2 -8582.355} C_VEL
LIN {X 0,Y 446.385,Z 696.883,A -85,B 0,C 180,E1 -8585.619,E2 -8585.619} C_VEL
LIN {X 0,Y 446.43,Z 696.864,A -85,B 0,C 180,E1 -8589.018,E2 -8589.018} C_VEL
LIN {X 0,Y 446.409,Z 696.876,A -85,B 0,C 180,E1 -8592.273,E2 -8592.273} C_VEL
LIN {X 0,Y 446.411,Z 696.866,A -85,B 0,C 180,E1 -8595.097,E2 -8595.097} C_VEL
LIN {X 0,Y 446.394,Z 696.878,A -85,B 0,C 180,E1 -8598.605,E2 -8598.605} C_VEL
LIN {X 0,Y 446.425,Z 696.87,A -85,B 0,C 180,E1 -8600.971,E2 -8600.971} C_VEL
LIN {X 0,Y 446.364,Z 696.881,A -85,B 0,C 180,E1 -8604.369,E2 -8604.369} C_VEL
LIN {X 0,Y 446.369,Z 696.88,A -85,B 0,C 180,E1 -8607.634,E2 -8607.634} C_VEL
LIN {X 0,Y 446.406,Z 696.87,A -85,B 0,C 180,E1 -8610.787,E2 -8610.787} C_VEL
LIN {X 0,Y 446.412,Z 696.877,A -85,B 0,C 180,E1 -8613.844,E2 -8613.844} C_VEL
LIN {X 0,Y 446.362,Z 696.879,A -85,B 0,C 180,E1 -8616.819,E2 -8616.819} C_VEL
LIN {X 0,Y 446.374,Z 696.879,A -85,B 0,C 180,E1 -8619.734,E2 -8619.734} C_VEL
LIN {X 0,Y 446.393,Z 696.875,A -85,B 0,C 180,E1 -8622.594,E2 -8622.594} C_VEL
LIN {X 0,Y 446.409,Z 696.875,A -85,B 0,C 180,E1 -8625.41,E2 -8625.41} C_VEL
LIN {X 0,Y 446.474,Z 696.867,A -85,B 0,C 180,E1 -8628.192,E2 -8628.192} C_VEL
LIN {X 0,Y 446.526,Z 696.86,A -85,B 0,C 180,E1 -8631.856,E2 -8631.856} C_VEL
LIN {X 0,Y 446.578,Z 696.859,A -85,B 0,C 180,E1 -8634.582,E2 -8634.582} C_VEL
LIN {X 0,Y 446.644,Z 696.849,A -85,B 0,C 180,E1 -8637.294,E2 -8637.294} C_VEL
LIN {X 0,Y 446.717,Z 696.838,A -85,B 0,C 180,E1 -8640,E2 -8640} C_VEL
LIN {X 0,Y 446.644,Z 696.845,A -85,B 0,C 180,E1 -8642.706,E2 -8642.706} C_VEL
LIN {X 0,Y 446.576,Z 696.855,A -85,B 0,C 180,E1 -8646.325,E2 -8646.325} C_VEL
LIN {X 0,Y 446.469,Z 696.868,A -85,B 0,C 180,E1 -8649.057,E2 -8649.057} C_VEL
LIN {X 0,Y 446.462,Z 696.869,A -85,B 0,C 180,E1 -8652.731,E2 -8652.731} C_VEL
LIN {X 0,Y 446.446,Z 696.869,A -85,B 0,C 180,E1 -8656.241,E2 -8656.241} C_VEL
LIN {X 0,Y 446.398,Z 696.88,A -85,B 0,C 180,E1 -8659.306,E2 -8659.306} C_VEL
LIN {X 0,Y 446.351,Z 696.882,A -85,B 0,C 180,E1 -8662.203,E2 -8662.203} C_VEL
LIN {X 0,Y 446.407,Z 696.874,A -85,B 0,C 180,E1 -8665.155,E2 -8665.155} C_VEL
LIN {X 0,Y 446.42,Z 696.876,A -85,B 0,C 180,E1 -8668.183,E2 -8668.183} C_VEL
LIN {X 0,Y 446.37,Z 696.877,A -85,B 0,C 180,E1 -8671.304,E2 -8671.304} C_VEL
LIN {X 0,Y 446.371,Z 696.88,A -85,B 0,C 180,E1 -8674.528,E2 -8674.528} C_VEL
LIN {X 0,Y 446.385,Z 696.875,A -85,B 0,C 180,E1 -8678.089,E2 -8678.089} C_VEL
LIN {X 0,Y 446.396,Z 696.877,A -85,B 0,C 180,E1 -8680.927,E2 -8680.927} C_VEL
LIN {X 0,Y 446.396,Z 696.879,A -85,B 0,C 180,E1 -8683.847,E2 -8683.847} C_VEL
LIN {X 0,Y 446.401,Z 696.88,A -85,B 0,C 180,E1 -8686.403,E2 -8686.403} C_VEL
LIN {X 0,Y 446.427,Z 696.875,A -85,B 0,C 180,E1 -8689.811,E2 -8689.811} C_VEL
LIN {X 0,Y 446.393,Z 696.881,A -85,B 0,C 180,E1 -8692.13,E2 -8692.13} C_VEL
LIN {X 0,Y 446.395,Z 696.874,A -85,B 0,C 180,E1 -8695.484,E2 -8695.484} C_VEL
LIN {X 0,Y 446.422,Z 696.951,A -85,B 0,C 180,E1 -8698.622,E2 -8698.622} C_VEL
LIN {X 0,Y 450.134,Z 713.08,A -85,B 0,C 180,E1 -8701.209,E2 -8701.209} C_VEL
LIN {X 0,Y 450.997,Z 717.454,A -85,B 0,C 180,E1 -8701.884,E2 -8701.884} C_VEL
LIN {X 0,Y 450.379,Z 731.46,A -85,B 0,C 180,E1 -8703.852,E2 -8703.852} C_VEL
LIN {X 0,Y 449.157,Z 756.094,A -85,B 0,C 180,E1 -8707.261,E2 -8707.261} C_VEL
LIN {X 0,Y 447.998,Z 781.586,A -85,B 0,C 180,E1 -8710.773,E2 -8710.773} C_VEL
LIN {X 0,Y 447.607,Z 791.413,A -85,B 0,C 180,E1 -8712.135,E2 -8712.135} C_VEL
LIN {X 0,Y 450.599,Z 819.218,A -85,B 0,C 180,E1 -8712.709,E2 -8712.709} C_VEL
LIN {X 0,Y 449.849,Z 902.263,A -85,B 0,C 180,E1 -8714.053,E2 -8714.053} C_VEL
LIN {X 0,Y 449.401,Z 915.502,A -85,B 0,C 180,E1 -8714.444,E2 -8714.444} C_VEL
LIN {X 0,Y 448.814,Z 928.834,A -85,B 0,C 180,E1 -8715.034,E2 -8715.034} C_VEL
LIN {X 0,Y 448.174,Z 940.066,A -85,B 0,C 180,E1 -8715.708,E2 -8715.708} C_VEL
LIN {X 0,Y 447.635,Z 951.134,A -85,B 0,C 180,E1 -8716.558,E2 -8716.558} C_VEL
LIN {X 0,Y 447.153,Z 962.404,A -85,B 0,C 180,E1 -8717.642,E2 -8717.642} C_VEL
LIN {X 0,Y 446.625,Z 971.078,A -85,B 0,C 180,E1 -8718.663,E2 -8718.663} C_VEL
LIN {X 0,Y 446.232,Z 979.113,A -85,B 0,C 180,E1 -8719.801,E2 -8719.801} C_VEL
LIN {X 0,Y 445.971,Z 986.996,A -85,B 0,C 180,E1 -8721.168,E2 -8721.168} C_VEL
LIN {X 0,Y 445.773,Z 994.277,A -85,B 0,C 180,E1 -8722.761,E2 -8722.761} C_VEL
LIN {X 0,Y 445.754,Z 999.144,A -85,B 0,C 180,E1 -8724.124,E2 -8724.124} C_VEL
LIN {X 0,Y 445.746,Z 1002.87,A -85,B 0,C 180,E1 -8725.485,E2 -8725.485} C_VEL
LIN {X 0,Y 445.772,Z 1004.795,A -85,B 0,C 180,E1 -8726.391,E2 -8726.391} C_VEL
LIN {X 0,Y 445.737,Z 1006.231,A -85,B 0,C 180,E1 -8727.295,E2 -8727.295} C_VEL
LIN {X 0,Y 445.738,Z 1007.257,A -85,B 0,C 180,E1 -8728.199,E2 -8728.199} C_VEL
LIN {X 0,Y 445.73,Z 1007.881,A -85,B 0,C 180,E1 -8729.103,E2 -8729.103} C_VEL
LIN {X 0,Y 445.734,Z 1008.102,A -85,B 0,C 180,E1 -8730.006,E2 -8730.006} C_VEL
LIN {X 0,Y 445.73,Z 1007.874,A -85,B 0,C 180,E1 -8730.909,E2 -8730.909} C_VEL
LIN {X 0,Y 445.739,Z 1007.245,A -85,B 0,C 180,E1 -8731.813,E2 -8731.813} C_VEL
LIN {X 0,Y 445.739,Z 1006.213,A -85,B 0,C 180,E1 -8732.717,E2 -8732.717} C_VEL
LIN {X 0,Y 445.776,Z 1004.771,A -85,B 0,C 180,E1 -8733.621,E2 -8733.621} C_VEL
LIN {X 0,Y 445.76,Z 1001.735,A -85,B 0,C 180,E1 -8734.98,E2 -8734.98} C_VEL
LIN {X 0,Y 445.754,Z 996.562,A -85,B 0,C 180,E1 -8736.639,E2 -8736.639} C_VEL
LIN {X 0,Y 445.872,Z 990.288,A -85,B 0,C 180,E1 -8738.161,E2 -8738.161} C_VEL
LIN {X 0,Y 446.09,Z 983.204,A -85,B 0,C 180,E1 -8739.527,E2 -8739.527} C_VEL
LIN {X 0,Y 446.493,Z 974.369,A -85,B 0,C 180,E1 -8740.893,E2 -8740.893} C_VEL
LIN {X 0,Y 446.909,Z 965.336,A -85,B 0,C 180,E1 -8742.032,E2 -8742.032} C_VEL
LIN {X 0,Y 447.458,Z 954.535,A -85,B 0,C 180,E1 -8743.143,E2 -8743.143} C_VEL
LIN {X 0,Y 448.014,Z 943.086,A -85,B 0,C 180,E1 -8744.078,E2 -8744.078} C_VEL
LIN {X 0,Y 448.667,Z 930.636,A -85,B 0,C 180,E1 -8744.868,E2 -8744.868} C_VEL
LIN {X 0,Y 449.232,Z 918.869,A -85,B 0,C 180,E1 -8745.429,E2 -8745.429} C_VEL
LIN {X 0,Y 449.728,Z 906.319,A -85,B 0,C 180,E1 -8745.847,E2 -8745.847} C_VEL
LIN {X 0,Y 450.047,Z 890.352,A -85,B 0,C 180,E1 -8746.156,E2 -8746.156} C_VEL
LIN {X 0,Y 450.496,Z 817.16,A -85,B 0,C 180,E1 -8747.327,E2 -8747.327} C_VEL
LIN {X 0,Y 447.626,Z 791.305,A -85,B 0,C 180,E1 -8747.878,E2 -8747.878} C_VEL
LIN {X 0,Y 448.679,Z 766.089,A -85,B 0,C 180,E1 -8751.362,E2 -8751.362} C_VEL
LIN {X 0,Y 449.878,Z 741.805,A -85,B 0,C 180,E1 -8754.706,E2 -8754.706} C_VEL
LIN {X 0,Y 451.041,Z 719.112,A -85,B 0,C 180,E1 -8757.874,E2 -8757.874} C_VEL
LIN {X 0,Y 450.36,Z 714.325,A -85,B 0,C 180,E1 -8758.595,E2 -8758.595} C_VEL
LIN {X 0,Y 446.428,Z 696.878,A -85,B 0,C 180,E1 -8761.39,E2 -8761.39} C_VEL
LIN {X 0,Y 446.369,Z 696.886,A -85,B 0,C 180,E1 -8764.533,E2 -8764.533} C_VEL
LIN {X 0,Y 446.398,Z 696.878,A -85,B 0,C 180,E1 -8767.884,E2 -8767.884} C_VEL
LIN {X 0,Y 446.411,Z 696.88,A -85,B 0,C 180,E1 -8771.397,E2 -8771.397} C_VEL
LIN {X 0,Y 446.431,Z 696.876,A -85,B 0,C 180,E1 -8775.111,E2 -8775.111} C_VEL
LIN {X 0,Y 446.416,Z 696.875,A -85,B 0,C 180,E1 -8778.607,E2 -8778.607} C_VEL
LIN {X 0,Y 446.415,Z 696.875,A -85,B 0,C 180,E1 -8781.926,E2 -8781.926} C_VEL
LIN {X 0,Y 446.437,Z 696.877,A -85,B 0,C 180,E1 -8785.478,E2 -8785.478} C_VEL
LIN {X 0,Y 446.428,Z 696.874,A -85,B 0,C 180,E1 -8788.701,E2 -8788.701} C_VEL
LIN {X 0,Y 446.464,Z 696.873,A -85,B 0,C 180,E1 -8791.832,E2 -8791.832} C_VEL
LIN {X 0,Y 446.453,Z 696.873,A -85,B 0,C 180,E1 -8794.847,E2 -8794.847} C_VEL
LIN {X 0,Y 446.464,Z 696.871,A -85,B 0,C 180,E1 -8798.246,E2 -8798.246} C_VEL
LIN {X 0,Y 446.466,Z 696.874,A -85,B 0,C 180,E1 -8801.65,E2 -8801.65} C_VEL
LIN {X 0,Y 446.464,Z 696.872,A -85,B 0,C 180,E1 -8802.582,E2 -8802.582} C_VEL
LIN {X 0,Y 450.879,Z 708.393,A -85,B 0,C 180,E1 -8803.06,E2 -8803.06} C_VEL
LIN {X 0,Y 450.086,Z 778.959,A -85,B 0,C 180,E1 -8804.432,E2 -8804.432} C_VEL
LIN {X 0,Y 449.966,Z 790.954,A -85,B 0,C 180,E1 -8804.805,E2 -8804.805} C_VEL
LIN {X 0,Y 449.832,Z 800.852,A -85,B 0,C 180,E1 -8805.235,E2 -8805.235} C_VEL
LIN {X 0,Y 449.573,Z 810.883,A -85,B 0,C 180,E1 -8805.796,E2 -8805.796} C_VEL
LIN {X 0,Y 449.26,Z 820.002,A -85,B 0,C 180,E1 -8806.429,E2 -8806.429} C_VEL
LIN {X 0,Y 448.853,Z 829.338,A -85,B 0,C 180,E1 -8807.223,E2 -8807.223} C_VEL
LIN {X 0,Y 448.561,Z 837.155,A -85,B 0,C 180,E1 -8808.018,E2 -8808.018} C_VEL
LIN {X 0,Y 448.212,Z 844.702,A -85,B 0,C 180,E1 -8808.926,E2 -8808.926} C_VEL
LIN {X 0,Y 447.785,Z 852.492,A -85,B 0,C 180,E1 -8810.058,E2 -8810.058} C_VEL
LIN {X 0,Y 447.478,Z 858.924,A -85,B 0,C 180,E1 -8811.192,E2 -8811.192} C_VEL
LIN {X 0,Y 447.198,Z 864.153,A -85,B 0,C 180,E1 -8812.297,E2 -8812.297} C_VEL
LIN {X 0,Y 446.89,Z 869.364,A -85,B 0,C 180,E1 -8813.68,E2 -8813.68} C_VEL
LIN {X 0,Y 446.624,Z 872.21,A -85,B 0,C 180,E1 -8814.582,E2 -8814.582} C_VEL
LIN {X 0,Y 446.466,Z 876.136,A -85,B 0,C 180,E1 -8816.39,E2 -8816.39} C_VEL
